StartSequence := FALSE;
b_ExtContactor := mode = eBreakerOperationMode.ExtGrid;
ton_ResetSEQ();

//SEQUENCER
CASE by_SequenceIndexes[ExecIndex] OF
	0: 	ExecIndex := 0; StartSequence := TRUE; by_RetryCounter := 0; by_CurrentStep := 0;
	1:	ton_ResetSEQ.IN := FALSE; by_CurrentStep := 1;
		b_trigger := Warmup(get.b_gensetHot);
	2:  b_trigger := SEL(b_ExtContactor, Inputcontactor.Close(b_SynchroneGenset OR b_GridFollowingMode), Extcontactor.Close(FALSE));
		get.e_state := eGenGridState.Synchronization; by_CurrentStep := 2;
		ton_ResetSEQ.IN := TRUE;
	3:	b_trigger := b_escapeCondition; by_CurrentStep := 3;
		get.e_state := eGenGridState.Starting;
END_CASE

ton_SeqPulse(IN := b_trigger AND NOT ton_SeqPulse.Q);
IF ton_SeqPulse.Q THEN
	ExecIndex := ExecIndex +1;
END_IF

IF ton_ResetSEQ.Q THEN
	ExecIndex := 0;
	ton_ResetSEQ.IN := FALSE;
	by_RetryCounter := by_RetryCounter + 1;
END_IF

IF by_RetryCounter > st_params.by_SyncRetries THEN
	by_RetryCounter := 0;
	get.events.b_WarmupFault := by_CurrentStep = 1;
	get.events.b_SynchronisationFault := by_CurrentStep = 2;
	get.events.b_StartupFault := by_CurrentStep = 3;
END_IF

//The exit from the current step. if breaker already closed, continue normal SFC procedure.
IF b_genOnly AND NOT b_startcondition AND NOT b_BreakerFb THEN
	b_IOStartStop := FALSE;
	SFCreset := TRUE;
END_IF
END_METHOD

METHOD StartStopConditions
VAR_INPUT
	enable			: BOOL;
END_VAR

VAR_INST
	r_LoadPercentOutput : REAL;
	b_Charging			: BOOL;
	r_InverterLoad		: REAL;
	r_InputLoad			: REAL;
	b_BatErrorGenStartTrigger : BOOL;
END_VAR
b_Charging:= monitor.powerstack.r_ActivePower < 0;
r_InverterLoad := monitor.powerstack.r_LoadPercent * SEL(b_Charging, 1, -1) * 0.97;// * monitor.system.r_CurrentEfficiency/100;
r_InputLoad	:= monitor.powermonitor.InputField.r_loadshare;
r_LoadPercentOutput := r_InputLoad + r_InverterLoad;

IF enable THEN
	ChargeLoadStart(
		enable:= b_loadbankEnable,
		reset := FALSE,
		value:= monitor.powerstack.r_LoadPercent, 
		startvalue:= MIN(GensetSetpoints.r_BatteryloadStart, monitor.powerstack.r_OvercurrentValueAct *100),
		stopvalue := GensetSetpoints.r_BatteryloadStop - monitor.powermonitor.InputField.r_loadshare,
		OffDelay := T#3M,
		OnDelay := T#10S);
	
	LoadStart(
		enable := monitor.powerstack.b_ControlEnabled,
		reset := r_LoadPercentOutput < -10,// if charging reset.
		value := r_LoadPercentOutput,
		StartValue:= MIN(GensetSetpoints.r_BatteryloadStart, monitor.powerstack.r_OvercurrentValueAct *100),
		StopValue :=  GensetSetpoints.r_BatteryloadStop,
		OffDelay := St_params.Genset.OverloadOffDelay,
		OnDelay := St_params.Genset.OverloadOnDelay,
		);
	
	SoCStart(
		enable := monitor.system.e_State <> eSystemState.Discharging_Only,
		reset := FALSE,
		value := monitor.battery.BatteryInfo.r_SOCScaled,
		StartValue:=  GensetSetpoints.r_SocStart,
		StopValue :=  MAX(GensetSetpoints.r_SocStop, GensetSetpoints.r_SocStart + 0.5));
		
	BatFullStart(
		enable:= b_loadbankEnable,
		reset := monitor.powerstack.r_ActivePower < -5 AND NOT b_loadbankEnable,
		value := monitor.battery.BatteryInfo.r_SOCScaled,
		StartValue:=  control.SoftSettings.system.r_SocMax,
		StopValue :=  control.SoftSettings.system.r_SocMax - settings.MachineParams.BMS.r_SocHysteresis,
		OffDelay := T#3M,
		OnDelay := T#10S
		);


ELSE
	BatFullStart(reset:= TRUE);
	SoCStart(reset := TRUE);
	LoadStart(reset := TRUE);
	ChargeLoadStart(reset := TRUE);
END_IF

//Trigger genset start when battery down.
IF NOT gensetsetpoints.b_StartAtBatteryError OR b_BESSready	THEN
	b_BatErrorGenStartTrigger := FALSE;
ELSIF NOT b_startcondition THEN
	b_BatErrorGenStartTrigger := TRUE;
END_IF

//Summerize conditions
b_StartCondition := ((LoadStart.Q OR SOCStart.Q OR BatFullStart.Q OR ChargeLoadStart.Q OR b_BatErrorGenStartTrigger) AND
						get.e_GensetStartStop= eGensetStartStop.Auto) OR 
						get.e_GensetStartStop= eGensetStartStop.Start;

//get run condition
IF get.e_GensetStartStop= eGensetStartStop.Start THEN
	get.e_RunCondition := eRunCondition.ManuallyStarted;
ELSIF get.e_GensetStartStop= eGensetStartStop.stop THEN
	get.e_RunCondition := eRunCondition.ManuallyStopped;
ELSIF SOCStart.Q THEN
	get.e_RunCondition := eRunCondition.SoC;	
ELSIF LoadStart.Q THEN
	get.e_RunCondition := eRunCondition.DischargeOverload;
ELSIF ChargeLoadStart.Q THEN
	get.e_RunCondition := eRunCondition.ChargeOverload;
ELSIF BatFullStart.Q THEN
	get.e_RunCondition := eRunCondition.BattFull;
ELSE
	get.e_RunCondition := eRunCondition.None;
END_IF
END_METHOD

ACTION STARTUP_active:
get.e_state := eGenGridState.Starting;
b_SFCmodetransInhibit := FALSE;
get.b_active := TRUE;


SFCtip := StartSequence(
			mode := BreakerOperationMode, 
			b_breakerfb := b_breakerFb,
			b_AcOK	:= b_BreakerACok,
			b_gridfollowingMode := b_GridACDetected,
			SFCreset => SFCResetTrigger
			) AND NOT sfctip;

//Reset before running again.		
GenDownCheck(FALSE, TRUE);
END_ACTION

ACTION STOP_active:
get.e_state := eGenGridState.Stopping;
SFCtransTrigger.in := FALSE;

CASE BreakerOperationMode OF
	eBreakerOperationMode.GenFix:
		IF Cooldown(TRUE) THEN SFCTransTrigger.in := InputContactor.Open(FALSE); END_IF
	eBreakerOperationMode.GenIso, eBreakerOperationMode.GenDroop:
	IF GenDownCheck(FALSE, FALSE) OR NOT b_breakerACOK THEN
		SFCTransTrigger.in := Inputcontactor.Open(TRUE) AND cooldown(TRUE);
	ELSIF NOT b_hybridMode AND b_startCondition AND monitor.powerstack.b_ControlEnabled AND NOT Get.b_ModeTransActive THEN
		InputContactor.Deload(TRUE);
		SFCTransTrigger.in := TRUE;
	ELSE
		SFCTransTrigger.in := InputContactor.Open(b_hybridMode) AND_THEN Cooldown(FALSE);
	END_IF
		
	eBreakerOperationMode.GridFeedthrough:
		IF b_AMFEnabled AND monitor.powerstack.b_ControlEnabled OR get.b_ModeTransActive THEN SFCTransTrigger.in := inputcontactor.Open(NOT Get.b_ModeTransActive OR get.events.b_CurrentLimitTrip);
		ELSE SFCTransTrigger.in := TRUE; END_IF
	eBreakerOperationMode.ExtGrid: 
		IF b_AMFEnabled AND monitor.powerstack.b_ControlEnabled THEN SFCTransTrigger.in := extcontactor.Open(control.SoftSettings.PSB.b_BreakerControl);
		ELSE SFCTransTrigger.in := TRUE; END_IF
END_CASE



SFCtip := SFCTransTrigger.Q AND NOT SFCtip;
END_ACTION

METHOD ThreePointSelector : REAL
VAR_INPUT
	r1max	: REAL;
	r2      : REAL;
	r3      : REAL;
	b2		: BOOL;
	b3		: BOOL;
END_VAR

VAR
	temp	: REAL;
END_VAR
IF b2 AND NOT b3 THEN
	temp := r2;
ELSIF NOT b2 AND b3 THEN
	temp := r3;
ELSE
	temp := r1max;
END_IF

ThreepointSelector := LIMIT(0,temp,r1max);
END_METHOD

ACTION WAITINGTRIGGER_active:
get.e_state := eGenGridState.Waiting_Trigger;
SFCTransTrigger.IN := FALSE;
get.b_active := FALSE;

CASE BreakerOperationMode OF
	eBreakerOperationMode.GenIso:
		SFCTransTrigger(IN := b_StartCondition AND NOT GenDownCheck(FALSE , b_StartCondition));
	eBreakerOperationMode.GenDroop:
		SFCTransTrigger(IN := b_StartCondition AND NOT GenDownCheck(FALSE , b_StartCondition)); 
	eBreakerOperationMode.Genfix:
		SFCTransTrigger(IN := b_StartCondition AND NOT GenDownCheck(FALSE , b_StartCondition) AND b_BESSReady AND b_BusbarACOK);
	eBreakerOperationMode.Gridfeedthrough, eBreakerOperationMode.ExtGrid: 
		SFCTransTrigger(IN := b_breakerACOK);
		get.e_state := eGenGridState.Waiting_For_AC;
		IF NOT GridOKdetect(FALSE) THEN
			get.e_state := eGenGridState.Gridcode_Release_Check;
			SFCTransTrigger.in := FALSE;
		END_IF
END_CASE

IF get.b_ModeTransActive THEN
	get.e_state := eGenGridState.Waiting_Mode_Reconnect;
END_IF

IF b_ForceOperate OR (b_breakerfb AND b_breakerACOK) THEN
	SFCTransTrigger.in := TRUE;
END_IF



//Trigger to start. Only if modeswitch is disabled.
SFCtip := SFCTransTrigger.Q AND NOT get.b_ModeTransActive AND NOT SFCtip AND NOT get.events.b_StartingInhibit;
END_ACTION

METHOD Warmup : BOOL
VAR_INPUT
	Skip		: BOOL;
END_VAR

VAR_INST
	t_time				: TIME;
	b_startfb			: BOOL;
	ton_StartTimeOut	: TON;
	tof_reset			: Tof := (PT:= T#20MS);
END_VAR
b_IOStartStop := TRUE;
Warmup := FALSE;

b_startFb := b_BreakerACok;
IF NOT b_breakerACOK THEN
	inputcontactor.open(TRUE);
	get.e_state := eGenGridState.Starting;
ELSE
	get.e_state := eGenGridState.Warmup;
END_IF

tof_reset(IN:= NOT ton_StartTimeOut.Q);
ton_StartTimeOut(IN := b_startfb AND tof_reset.Q, PT:= t_WarmupTime); 

IF ton_StartTimeOut.Q OR skip THEN
	get.b_gensetHot := TRUE;
	ton_StartTimeOut.IN := FALSE;
	Warmup := b_IOStartStop;
END_IF
END_METHOD

METHOD ZeroCurrentDisconnect : BOOL
VAR_INPUT
END_VAR

VAR_INST
	ton_FlatZeroCurrentTimeOut 	: TON := (PT:= T#50MS);
END_VAR
ton_FlatZeroCurrentTimeOut(
	IN := TO_INT(ar_BreakerCurrent[phases.L1]) = 0 OR TO_INT(ar_BreakerCurrent[phases.L2]) = 0 OR TO_INT(ar_BreakerCurrent[phases.L3]) = 0,
	Q => ZeroCurrentDisconnect);
END_METHOD

END_FUNCTION_BLOCK

// ---- POUs/System/GenGridControl/FB_ContactorControl.TcPOU
FUNCTION_BLOCK FB_ContactorControl
VAR_IN_OUT CONSTANT
	monitor								   	: ST_System_Monitor;
	control									: ST_System_Control;
	st_params								: ST_ContactorControl_params;
END_VAR

VAR_IN_OUT
	SyncData								: ST_GenGridController_SyncData;

END_VAR

VAR_INPUT
	b_fbIn			: BOOL;
	b_deadbus		: BOOL;
	b_SyncOK		: BOOL;
	li_VoltCrossRef	: LINT;
	li_VoltCrossBus	: LINT;
	r_AcVoltageRef	: REAL;
	r_AcFreqRef		: REAL;
	e_AcRotationRef : eACRotationState; // Fsource of reference
	e_AcRotationBus	: eACRotationState; //bus 
	ar_current		: ARRAY [0..4] OF REAL;
	r_power			: REAL;	
	b_deloadEnable	: BOOL;
END_VAR
VAR_OUTPUT
	CloseCMD		: BOOL;
	OpenCMD			: BOOL;
	SyncEnable		: BOOL;
	FreqSet			: REAL;
	VoltSet			: REAL;
	ACok			: BOOL;	
	b_fb			: BOOL;
	b_Deload		: BOOL;
	RotationFault	: BOOL;
END_VAR

VAR
	ton_SyncDelay 	: TON := (PT:=  T#1S);
	
	ton_synccheckoffdelay : TON := (PT :=T#1s);
	SyncCheck		: BOOL;
	fb_VoltPID			: FB_CTRL_PID_EXT;
	st_Params_VoltPID				: ST_CTRL_PID_EXT_PARAMS := ( 
										tTaskCycleTime := T#1MS,
										tCtrlCycleTime := T#1MS,
										fKp	:= 0.3,
										tTn := T#200MS,
										tTd := T#0MS,
										tTv := T#0MS,
										fOutMaxLimit := 40,
										fOutMinLimit := -40										
);
END_VAR

ACok := ACcheck(r_voltage := r_ACVoltageRef, r_frequency := r_ACFreqRef);
CheckRotationField();
SyncEnable := syncdata.b_Sync OR SyncCheck;
ton_SyncDelay(IN := SyncEnable);
b_fb := b_fbIn;

fb_VoltPID(stParams := st_Params_VoltPID);
ton_synccheckoffdelay(IN:= b_fb);
IF ton_synccheckoffdelay.Q THEN
	synccheck := FALSE;
	fb_VoltPID.eMode:= e_Ctrl_mode.eCTRL_MODE_RESET;
END_IF

METHOD CheckRotationField : BOOL
VAR_INPUT
END_VAR
IF e_ACRotationRef <> 0 AND e_ACRotationBus <> 0 THEN // if both are connected to AC
	IF e_ACRotationRef = e_ACRotationBus THEN
		CheckRotationField := TRUE;
		RotationFault := FALSE;
	ELSE
		RotationFault := TRUE;
	END_IF
ELSE
	RotationFault := FALSE;
END_IF
END_METHOD

METHOD Close : BOOL
VAR_INPUT
	Force	: BOOL;
END_VAR
VAR_INST
	ton_ACOKrelease : TON := (PT:= T#1S); 
	b_VoltageDetected	: BOOL;
	
	ton_SyncOK			: TON := (PT := T#5S);
END_VAR
ton_ACOKrelease(IN:= ACok);
b_VoltageDetected := r_ACVoltageRef > 100;
OpenCMD := FALSE;
syncCheck := FALSE;

ton_SyncOK(IN :=b_syncOK);
IF b_fbIN OR b_deadbus THEN
	CloseCMD := TRUE;
ELSIF force THEN
	IF b_VoltageDetected AND NOT b_deadbus THEN
		syncCheck := TRUE;
		CloseCMD := ton_SyncOK.Q AND ton_ACOKrelease.Q;
	ELSE
		CloseCMD := TRUE;
	END_IF
ELSE
	CloseCMD:= Sync();
END_IF

Close := b_fbIN;
IF b_fbIN THEN
	Syncdata.b_Sync := FALSE;
	syncCheck := FALSE;
	ton_SyncOK.IN := FALSE;
	ton_ACOKrelease.IN :=  FALSE;
END_IF
END_METHOD

METHOD Deload : BOOL
VAR_INPUT
	reset : BOOL;
END_VAR

VAR_INST
	release : BOOL;
	PowerReleaseThreshold : REAL;
	
END_VAR
IF b_deloadEnable AND NOT reset THEN
	b_Deload := TRUE;
	PowerReleaseThreshold := st_params.ui_DeloadCurrentRelease * r_AcVoltageRef *  1.73 / 1000; 
	release := ABS(ar_current[0]) < st_params.ui_DeloadCurrentRelease OR ABS(r_power) < (PowerReleaseThreshold);
	IF release THEN
		Deload := TRUE;
	END_IF
ELSE
    b_Deload := FALSE;
	Deload := TRUE;
END_IF
END_METHOD

METHOD FreqControlPID : BOOL;
VAR_INPUT
	r_ACRef				: REAL;
	r_ACintern			: REAL;
END_VAR

VAR_OUTPUT
	Q					: REAL;
END_VAR


VAR_INST
	r_phaseTimeDelta		: REAL;
	r_PeriodTime			: REAL;
	r_phaseAngle			: REAL;
	Buffer  				: ARRAY[0..2] OF REAL;
    Index   				: UINT := 0;
	di_tempAngle			: DINT;
	r_phaseAngleEMA        	: REAL := 0.0; // startwaarde
    Alpha       			: REAL := 0.5; // dempingsfactor tussen 0 en 1
	
		fb_FreqPID						: FB_CTRL_PID_EXT;
		st_Params_FreqPID				: ST_CTRL_PID_EXT_PARAMS := ( 
										tTaskCycleTime := T#1MS,
										tCtrlCycleTime := T#1MS,
										fKp	:= 0.1,
										tTn := T#20MS,
										tTd := T#0MS,
										tTv := T#0MS,
										fOutMaxLimit := 0.03,
										fOutMinLimit := -0.03										
);
	ton_SyncOKdelay						: TON := (PT := T#1S);
	r_syncOKAngle						: REAL := 2.0;
	r_FreqOffset 						: REAL := -0.05;
	
	li_voltcrossbusLast					: LINT;
	li_VoltCrossRefLast					: LINT;
	ton_FreqPIDBypass					: TON := (PT := T#2S);
	
END_VAR
ton_FreqPIDBypass(IN := li_voltcrossbusLast = li_voltcrossbus OR li_VoltCrossRefLast = li_VoltCrossRef);
IF ton_FreqPIDBypass.Q THEN
	 r_freqOffset := -0.05;
	 ton_SyncOKdelay(IN := b_syncOK, PT:= T#0S);
ELSE
	r_PeriodTime := SEL(r_ACintern = 0, 1/r_ACintern, 0) * 1000;
	r_phaseTimeDelta := TO_REAL((li_VoltCrossbus - li_VoltCrossRef) MOD TO_DINT(r_PeriodTime*1000000)) /1000000;
	
	IF r_phaseTimeDelta > (r_PeriodTime /2)  THEN
		r_phaseTimeDelta := r_phaseTimeDelta - r_PeriodTime; 
	ELSIF r_phaseTimeDelta < -(r_PeriodTime /2) THEN
		r_phaseTimeDelta := r_phaseTimeDelta + r_PeriodTime; 
	END_IF
	
	// Stap 1: bereken eerst de DINT-waarde veilig
	di_tempAngle := TO_DINT(r_phaseTimeDelta * r_ACintern * 360);
	
	// Stap 3: schaal naar REAL
	r_phaseAngle := TO_REAL(di_tempAngle MOD 360000) / 1000;
	
	//setup filtering (median and exponential moving average)
	Buffer[Index MOD 3] := r_phaseAngle;
	Index := Index + 1;
	r_phaseAngleEMA := Alpha * median(buffer) + (1.0 - Alpha) * r_phaseAngleEMA;
	
	fb_FreqPID(
		fSetpointValue := 0,
		fActualValue :=  r_phaseAngleEMA,
		stParams:= st_Params_FreqPID,
		fout => r_FreqOffset);
		
	fb_FreqPID.bHold := r_phaseAngleEMA > 170 OR r_phaseAngleEMA < -170;
	
		
	IF NOT fb_FreqPID.bError THEN
		fb_FreqPID.eMode := e_CTRL_MODE.eCTRL_MODE_ACTIVE;
	ELSE
		fb_FreqPID.eMode := e_CTRL_MODE.eCTRL_MODE_RESET;
	END_IF
	
	ton_SyncOKdelay(IN := ABS(r_phaseAngleEMA) < r_syncOKAngle, PT:= T#2S);
END_IF

//set outputs
Q := r_ACRef - r_freqOffset;
FreqControlPID := ton_SyncOKdelay.Q;


//update on change values
li_voltcrossbusLast := li_voltcrossbus;
li_voltcrossrefLast := li_voltcrossref;
END_METHOD

METHOD FrequencyControl : BOOL
VAR_INPUT
	r_ACRef				: REAL;
	r_ACintern			: REAL;
END_VAR

VAR_OUTPUT
	Q					: REAL;
END_VAR


VAR_INST
	OK					: BOOL;
	r_FreqOffset 		: REAL := 0.1; // hz
END_VAR
//Go below ref Frequency.

Q := r_ACRef + r_FreqOffset;
OK := ABS(r_ACintern - r_ACRef) < ABS(4* r_FreqOffset);
FrequencyControl := OK;
END_METHOD

METHOD init : BOOL
VAR_INPUT
END_VAR
syncCheck := FALSE;
END_METHOD

METHOD Open : BOOL
VAR_INPUT
	b_force : BOOL;
END_VAR

VAR_INST
	ton_TimeOut : TON;
END_VAR
ton_TimeOut(PT := TO_TIME(TO_REAL(st_params.ui_DeloadTimeOut)*1000));
CloseCMD := FALSE;

IF b_force OR ton_timeOut.Q THEN
	OpenCMD := TRUE;
ELSE
	ton_TimeOut.IN := TRUE;
	OpenCMD := Deload(FALSE);
END_IF

open := NOT b_FbIN;
IF NOT b_fbIn THEN
	//Syncdata.b_Sync:= FALSE;
	ton_TimeOut.IN := FALSE;
	b_deload := FALSE;
	OpenCMD := FALSE;
END_IF
END_METHOD

METHOD PRIVATE Sync : BOOL

VAR_INST
	//OK : BOOL;
	phasecontrol : BOOL := FALSE;
	SyncOKSum	: BOOL;
	tp_SyncOK : TP := (PT := T#100MS);
END_VAR
Syncdata.b_Sync := ACok;

IF phasecontrol THEN //new method beckhoff phase matching
	SyncOKsum := FreqControlPID(r_ACFreqRef, monitor.powerstack.r_FrequencyD7, Q => Syncdata.r_freqSet);
ELSE //old method
	SyncOKSum := b_syncOK AND FrequencyControl(r_acRef := r_ACFreqRef,  r_ACintern := monitor.powerstack.r_FrequencyD7, Q => Syncdata.r_freqSet);
END_IF

tp_SyncOK(IN:= SyncOKsum AND
	ACok AND
	CheckRotationField() AND
	VoltageControl(r_acRef := r_ACvoltageRef, r_ACintern := monitor.powerstack.r_ACVoltageD7, Q => Syncdata.r_VoltSet)
	);

IF ton_SyncDelay.Q AND tp_SyncOK.Q THEN
	SyncOKSum := FALSE;
	Sync := TRUE;
END_IF
END_METHOD

METHOD VoltageControl : BOOL
VAR_INPUT
	r_ACRef				: REAL;
	r_ACintern			: REAL;
END_VAR
VAR_OUTPUT
	Q : REAL;
END_VAR

VAR_INST
	
	OK			: BOOL;
	VoltDev		: REAL;

END_VAR
//Go equal to ref voltage.
VoltDev := r_ACintern - r_ACRef; 

//TOTAL AC CURRENT LIMIT
st_Params_VoltPID.fInnerWindow :=  st_Params.VoltagePID.InnerWindow;
st_Params_VoltPID.fOuterWindow := st_Params.VoltagePID.OuterWindow;
st_Params_VoltPID.fKp := st_params.VoltagePID.Kp;
st_Params_VoltPID.tTn := TO_TIME(st_params.VoltagePID.Tn);
st_Params_VoltPID.tTd := TO_TIME(st_params.VoltagePID.Td);
st_Params_VoltPID.tTv := TO_TIME(st_params.VoltagePID.Tv);
st_params_VoltPID.fDeadBandInput := st_Params.VoltagePID.InputDeadband;
st_params_VoltPID.fDeadBandOutput := st_Params.VoltagePID.OutputDeadband;

fb_VoltPID.fActualValue := VoltDev;
	
IF st_Params.VoltagePID.enable THEN
	fb_VoltPID.eMode := e_CTRL_MODE.eCTRL_MODE_ACTIVE;
ELSE
	fb_VoltPID.eMode := e_CTRL_MODE.eCTRL_MODE_RESET;
END_IF
	
OK := ABS(VoltDev) < st_params.ui_VoltageDevSyncOK;
Q := r_ACRef + fb_VoltPId.fOut;
VoltageControl := OK;
END_METHOD

END_FUNCTION_BLOCK

// ---- POUs/Functions-FBs-Programs/_acFunctions/AcCheck.TcPOU
FUNCTION AcCheck : BOOL
VAR_INPUT
	r_Voltage	: REAL;
	r_Frequency	: REAL;
END_VAR

AcCheck	:= AcFrequencyCheck(r_Frequency) AND AcVoltageCheck(r_Voltage);

END_FUNCTION

// ---- POUs/Functions-FBs-Programs/_acFunctions/ACFrequencyCheck.TcPOU
FUNCTION ACFrequencyCheck : BOOL
VAR_INPUT
	IN			: REAL;
END_VAR
VAR
	r_min		: REAL;
	r_max		: REAL;
END_VAR

r_min:= settings.GridParams.r_GridFrequencyMin;
r_max:= settings.GridParams.r_GridFrequencyMax;

ACfrequencyCheck := LIMIT(r_min, IN, r_max) = IN;

END_FUNCTION

// ---- POUs/Functions-FBs-Programs/_acFunctions/ACVoltageCheck.TcPOU
FUNCTION ACVoltageCheck : BOOL
VAR_INPUT
	IN			: REAL;
END_VAR
VAR
	r_min		: REAL;
	r_max		: REAL;
END_VAR

r_min:= settings.GridParams.r_GridVoltageMin - 10;
r_max:= settings.GridParams.r_GridVoltageMax;

ACVoltageCheck := LIMIT(r_min, IN, r_max) = IN;

END_FUNCTION

// ---- POUs/Functions-FBs-Programs/_generalFunctions/Median.TcPOU
FUNCTION Median : REAL
VAR_IN_OUT
    arr : ARRAY[*] OF REAL;
END_VAR

VAR
    sorted : ARRAY[0..6] OF REAL;
    i, j   : INT;
    temp   : REAL;
    len    : INT;
END_VAR



// bepaal lengte
len := TO_INT(UPPER_BOUND(arr, 1) - LOWER_BOUND(arr, 1) + 1);

// safety check
IF len > 7 THEN
    len := 7;
END_IF

// kopie
FOR i := 0 TO len - 1 DO
    sorted[i] := arr[i + LOWER_BOUND(arr,1)];
END_FOR

// sort
FOR i := 0 TO len - 2 DO
    FOR j := 0 TO len - i - 2 DO
        IF sorted[j] > sorted[j + 1] THEN
            temp := sorted[j];
            sorted[j] := sorted[j + 1];
            sorted[j + 1] := temp;
        END_IF
    END_FOR
END_FOR

// median
IF (len MOD 2) = 0 THEN
    Median := (sorted[len/2 - 1] + sorted[len/2]) * 0.5;
ELSE
    Median := sorted[len/2];
END_IF

END_FUNCTION

// ---- POUs/Functions-FBs-Programs/_generalFunctions/FB_StartStop.TcPOU
FUNCTION_BLOCK FB_StartStop
VAR_INPUT
	enable : BOOL;
	reset: BOOL;
	value : REAL;
	StartValue : REAL;
	StopValue : REAL;
	GreaterThan	: BOOL;
	OffDelay	: TIME;
	OnDelay		: TIME;	
END_VAR
VAR_OUTPUT
	Q : BOOL;
END_VAR
VAR
	SR_Started : SR;
	ton_set : TON;
	ton_reset: TON;
	ton_minruntime : TON;
END_VAR

ton_set(PT := Ondelay);
ton_reset(PT := Ondelay);
ton_minruntime(PT := OffDelay);
SR_Started();

IF GreaterThan THEN
	ton_set.IN:= value >= StartValue AND NOT reset;
	ton_reset.IN:= value <= StopValue OR reset;
ELSE
	ton_set.IN:= value <= StartValue AND NOT reset;
	ton_reset.IN:= Value >= StopValue OR reset;
END_IF

ton_minruntime(IN:= sr_started.Q1);
IF enable THEN
	SR_Started.SET1 := ton_set.Q;
	SR_Started.RESET := ton_reset.Q AND ton_minruntime.Q;
	Q := sr_started.Q1;	
ELSE
	SR_Started.SET1 := FALSE;
	SR_Started.RESET := TRUE;
	Q := FALSE;
END_IF

END_FUNCTION_BLOCK

// ---- POUs/Functions-FBs-Programs/_generalFunctions/PackWord.TcPOU
FUNCTION PackWord : WORD
VAR_INPUT
	b0			: BOOL;
	b1			: BOOL;
	b2			: BOOL;
	b3			: BOOL;
	b4			: BOOL;
	b5			: BOOL;
	b6			: BOOL;
	b7			: BOOL;
	b8			: BOOL;
	b9			: BOOL;
	b10			: BOOL;
	b11			: BOOL;
	b12			: BOOL;
	b13			: BOOL;
	b14			: BOOL;
	b15			: BOOL;
END_VAR

PackWord.0	:= b0;
PackWord.1	:= b1;
PackWord.2	:= b2;
PackWord.3	:= b3;
PackWord.4	:= b4;
PackWord.5	:= b5;
PackWord.6	:= b6;
PackWord.7	:= b7;
PackWord.8	:= b8;
PackWord.9	:= b9;
PackWord.10	:= b10;
PackWord.11	:= b11;
PackWord.12	:= b12;
PackWord.13	:= b13;
PackWord.14	:= b14;
PackWord.15	:= b15;

END_FUNCTION

// ---- POUs/Objects/ACDCCharger/FB_AcDcCharger.TcPOU
FUNCTION_BLOCK FB_AcDcCharger

VAR_IN_OUT CONSTANT
	st_params				:	ST_ACDCCharger_Params;
END_VAR

VAR_IN_OUT
	st_service : ST_ACDCCharger_Service;
END_VAR

VAR_INPUT
	enable					: 	BOOL;

	Set						:	ST_ACDCCharger_set;
	//BMS					:	st_BMS_BatterySummary;	
	r_Soc 					: 	REAL;
	r_SystemVoltage			: 	REAL;
	r_SystemCurrent			: 	REAL;
	r_MaxChargeCurrent		:	REAL;
	b_BatteryFullyCharged	: BOOL;
	b_BatteryOn				: BOOL;	
END_VAR
VAR_OUTPUT
	Get			:	ST_ACDCCharger_get;
	IPSRequest	:	ST_InternalPowerSupply_PowerDemand;
END_VAR
VAR
	BuscouplerState	AT %I*	: UINT;
	RxQueue			AT %I*	:	CANRXQUEUESTRUCT_E_10;  //without Transaction Time
	TxQueue			AT %Q*	:	CANTXQUEUESTRUCT_E_10;
	b_BuscouplerFound: BOOL;
END_VAR
VAR   // should add as input var
    bEmergencyStop : BOOL := FALSE;
    bResetFault : BOOL;
	GroupID	: BYTE := 1;
//	uiNumberofUnits	: UINT :=1;  // the number of units that are phyzicaly designed
//	rPset	: REAL; // AC Power set limit
//	rIset   : REAL; // AC Current set limit
//	bPowerMode : BOOL; // P mode sett selection
END_VAR
VAR	
	diag 	: ST_SystemDiagnostic;
    txIndex : INT;
    Step 	: INT;
    NumberOfMessagesToSend : INT := 10;

    voltage_mV : UDINT;
    current_mA : UDINT;
	stData : ST_Data;
    stControl : ST_Control;
	DeviceNo   : BYTE := 16#0B;
	rxIndex : INT; 
//    ChargerState : E_ChargerState := E_ChargerState.Idle;
	rVoltageWindow : REAL := 5.0;   // should be base on percentage or Volt?!
    bVoltageWindowOk : BOOL;  // check if voltage within the window
    b_ModuleCommunicationLost : BOOL;
    bWarning : BOOL;
    rChargerVoltageSetpoint : REAL;
    rChargerCurrentSetpoint : REAL;
    eval : ST_SystemEval;	
	bValidPrev : ARRAY [0..10] OF BOOL;  // test
	bFreezeCurrent : BOOL; // test	
	rMaxLimit		: REAL;

    tCycle : TON;
    tCheck : TON;
    tComWatchdog : TON;
    rPower_kW : REAL;
    rIsetReq : REAL := 60.0; (* configurable *)
    rCurrentCmd : REAL;
END_VAR
VAR CONSTANT
	e_ID 				: eObject_ID := eObject_ID.ACDCCharger;
END_VAR


IF enable THEN
	IF (BuscouplerState <> 8) THEN
		get.e_SystemStatus := eACDCChargerstate.init;
		get.Events.b_BuscouplerNotFound := TRUE;
	ELSE
		get.Events.b_BuscouplerNotFound := False;
		IF get.e_SystemStatus = eACDCChargerstate.init THEN
			get.e_SystemStatus := eACDCChargerstate.off;
		END_IF
		
		// should be 50ms to 200ms 
		tCycle(IN := NOT tCycle.Q, PT := T#50MS);
				
		IF tCycle.Q THEN
			ReadingRx();
			//UpdateStData();  // keep the last value! Useless?!
			EvaluateSystem();
			ChargingControl();
			SafetyCheck();
		    ValidateOutput();
			RunStateMachine();
			HandleCanCommunication();
			EvaluateDiagnostics();
		END_IF
	END_IF
END_IF

METHOD BuildCanId : DWORD
VAR_INPUT
    CommandNo  : BYTE;   // protocol command
    TargetAddr : BYTE := 1;   // group / module / broadcast(0x3F)
	
END_VAR
VAR
	 ErrorCode : BYTE := 0;   // always 0
	 SourceAddr : BYTE := 16#F0;   // Controller address
END_VAR

  // TargetAddr := 1;
   DeviceNo := 16#0B;
   ErrorCode:= 0;
   SourceAddr := 16#F0;
   
   
   BuildCanId :=
      SHL(DWORD#1,31)                // bit31 = extended CAN frame
   OR SHL(TO_DWORD(ErrorCode),26)       // error code
   OR SHL(TO_DWORD(DeviceNo),22)        // device number   Multicas: 0x0B, BroadCasti:0x0A
   OR SHL(TO_DWORD(CommandNo),16)       // command 
   OR SHL(TO_DWORD(TargetAddr),8)       // target address
   OR TO_DWORD(SourceAddr);             // source address
END_METHOD

METHOD PRIVATE ChargingControl
VAR_INPUT
END_VAR
VAR_INST
	rRawV : REAL;
	rPrevV : REAL;
	rRampLimitV : REAL := 20;
	rCurrentReq : REAL;
	rVoltageRamp : REAL;
	rAcPower	: REAL;
	rAcCurrent : REAL := 0.0;
	rMinGridVoltage	: REAL;
	i : INT;
	rTempMin : REAL;
	tDelayJumpOff	: TOf;
	bTestb : BOOL;
	srTest	: SR;
	tTestB : TOF;
	iUnitsTemp	: INT;
	
	iPrevHealthyModules : INT;
	tNewModuleTimer : TON;
	iEffectiveModules : INT;
	
	rTest : REAL;
	
	r_MinGridVoltageDerating 	: REAL := 1;
	r_TempDerating 				: REAL := 1;
	BMSChargeCurrentLimit		:	REAL;
	
	
END_VAR
 
// Battery Voltage from BMS

set.r_MinGridVoltage 	:= LIMIT(360, set.r_MinGridVoltage, 440);
set.r_currentSetpoint 	:= LIMIT(0, set.r_currentSetpoint, 125);
set.r_powersetpoint 	:= LIMIT(0, set.r_powersetpoint, st_params.ui_ModuleDesignPower * st_params.ui_NrOfInstalledModules);
set.r_SocTarget 		:= LIMIT(0, set.r_SocTarget, 100);

IF b_BatteryOn THEN // bms.e_BMS_PowerOnStatus = ePowerOnSTatus.On THEN
	rChargerVoltageSetpoint := r_SystemVoltage + st_params.r_VoltageWindow;
ELSE
	rChargerVoltageSetpoint := 0.0;
END_IF

IF r_Soc >= set.r_SocTarget OR b_BatteryFullyCharged THEN//bms.e_BMS_Status = eBMS_status.FullCharge THEN
	get.events.b_SOCLimitReached := TRUE;
ELSIF r_Soc < set.r_SocTarget - st_params.SocHysteresis THEN
	get.events.b_SOCLimitReached := FALSE;
END_IF


//rPower_kW := (stData.rSystemOutVoltageDc * stData.rSystemOutCurrentDc) / 1000.0;

rMinGridVoltage := 1000.0;
FOR i := 0 TO TO_INT(st_params.ui_NrOfInstalledModules - 1) DO
    IF stData.stModuleData[i].rExternalVoltageDc > 550 AND NOT stData.stModuleData[i].stStatus.bPfcOff  THEN
        
        rTempMin := MIN( stData.stModuleData[i].rVoltageL1L2,
            				stData.stModuleData[i].rVoltageL2L3,
            				stData.stModuleData[i].rVoltageL3L1 );
        
        rMinGridVoltage := MIN(rMinGridVoltage, rTempMin);        
    END_IF;
END_FOR;

IF (stData.rSystemOutVoltageDc > 1.0) THEN
	CASE set.e_ControlType OF
		ePowerControlType.Power		:	
			rIsetReq := (set.r_powersetpoint * 1000 / stData.rSystemOutVoltageDc) * 0.95;
			get.events.b_CurrentLimitActive := FALSE;
			
		ePowerControlType.Current 	:	
			rIsetReq := ((rMinGridVoltage * set.r_currentSetpoint * 1.73) / stData.rSystemOutVoltageDc) * 0.95;
			get.events.b_CurrentLimitActive := TRUE;
			
		ePowerControlType.Both 		:	
			rIsetReq := (set.r_powersetpoint * 1000 / stData.rSystemOutVoltageDc) * 0.95;
			IF (rMinGridVoltage * set.r_currentSetpoint * 1.73) < set.r_powersetpoint * 1000 THEN
				rIsetReq := ((rMinGridVoltage * set.r_currentSetpoint * 1.73) / stData.rSystemOutVoltageDc) * 0.95;
				get.events.b_CurrentLimitActive := TRUE;
			ELSE
				get.events.b_CurrentLimitActive := FALSE;
			END_IF
	END_CASE
ELSE
	riSetReq := 0;
END_IF

BMSChargeCurrentLimit := ABS(r_MaxChargeCurrent) + r_SystemCurrent + stData.rSystemOutCurrentDc;
IF BMSChargeCurrentLimit < rIsetReq THEN
	rCurrentCmd := BMSChargeCurrentLimit - 2;
	get.Events.b_BatteryLimitDeratingActive := TRUE;
ELSE
	rCurrentCmd := MIN(rCurrentCMD + ST_Params.BMSChargeLimitRampRate, rIsetReq);
	get.Events.b_BatteryLimitDeratingActive := FALSE;
END_IF

 
//ACVoltageRamp
IF rMinGridVoltage < set.r_MinGridVoltage THEN
	r_MinGridVoltageDerating := MAX(r_MinGridVoltageDerating * 0.999, 0.1);
ELSIF rMinGridVoltage > set.r_MinGridVoltage + st_params.GridVoltageHysteresis THEN
	r_MinGridVoltageDerating := MIN(r_MinGridVoltageDerating * 1.001, 1);
END_IF

get.Events.b_ACUnderVoltageDeratingActive := r_MinGridVoltageDerating < 1;


IF eval.rMaxTemperature > 80.0 THEN
	r_TempDerating := MAX(r_TempDerating * 0.999, 0.1);
ELSIF eval.rMaxTemperature < 75.0 THEN
	r_TempDerating := MIN(r_TempDerating * 1.001, 1);
END_IF
get.Events.b_TemperatureDeratingActive := r_TempDerating < 1;


// a unit back after a short lost( less than 10s  and keep stData.rNumberOfModules as original value)
iEffectiveModules := eval.iHealthyModules;
IF eval.iHealthyModules > iPrevHealthyModules THEN
	iEffectiveModules := eval.iHealthyModules + (eval.iHealthyModules - iPrevHealthyModules);
END_IF


// Current setpoint
//rCurrent := LIMIT(0.0, rCurrentCmd, eval.rTotalAvailableCurrent) / MAX(iEffectiveModules, 1);
IF bFreezeCurrent THEN
    rChargerCurrentSetpoint := 0;              // or keep last value if you prefer
    bFreezeCurrent := FALSE;    // only 1 cycle
ELSE
    rChargerCurrentSetpoint := LIMIT(0.0, rCurrentCmd, eval.rTotalAvailableCurrent) / MAX(iEffectiveModules, 1);
END_IF

iPrevHealthyModules := eval.iHealthyModules;

// if any unit is back after a long lost, stData.rNumberOfModules become 0 for a momment
tDelayJumpOff(IN := (stData.rNumberOfModules < eval.iHealthyModules), PT := T#1S);

IF tDelayJumpOff.Q THEN
	rChargerCurrentSetpoint := 0.0;
END_IF

IF iEffectiveModules > 0 THEN
	rChargerCurrentSetpoint := 
		LIMIT(0, rChargerCurrentSetpoint * r_MinGridVoltageDerating * r_TempDerating, eval.rTotalAvailableCurrent / iEffectiveModules);
ELSE
	rChargerCurrentSetpoint := 0;
END_IF
END_METHOD

METHOD EMSTOP : BOOL
VAR_INPUT
END_VAR


get.e_SystemStatus := eACDCChargerState.Fault;

EMSTOP := true;
END_METHOD

METHOD PRIVATE EvaluateDiagnostics
VAR
    i : INT;
END_VAR
	

//Reset all
diag.bAnyError 				:= FALSE;
diag.bAnyWarning 			:= FALSE;

diag.bError_OutputOV 		:= FALSE;
diag.bError_OverTemp 		:= FALSE;
diag.bError_ShortCircuit	:= FALSE;
diag.bError_ModuleError 	:= FALSE;
diag.bError_CommLost 		:= FALSE;
diag.bError_PhaseLost 		:= FALSE;

diag.bWarn_InputOV 			:= FALSE;
diag.bWarn_InputUV 			:= FALSE;
diag.bWarn_FanError 		:= FALSE;
diag.bWarn_PowerLimit 		:= FALSE;
diag.bWarn_TempHigh 		:= FALSE;

diag.bAllModulesOff 		:= TRUE;
diag.bAllModulesOn 			:= TRUE;


FOR i := 0 TO TO_INT(st_params.ui_NrOfInstalledModules - 1) DO

    //ERRORS
    IF stData.stModuleData[i].stStatus.bOutputOverVoltage THEN
        diag.bError_OutputOV := TRUE;
    END_IF

    IF stData.stModuleData[i].stStatus.bTempHigh THEN
        diag.bError_OverTemp := TRUE;
    END_IF

    IF stData.stModuleData[i].stStatus.bOutputShortCircuit THEN
        diag.bError_ShortCircuit := TRUE;
    END_IF

    IF stData.stModuleData[i].stStatus.bModuleError OR
       stData.stModuleData[i].stStatus.bModuleProtection THEN
        diag.bError_ModuleError := TRUE;
    END_IF

    IF stData.stModuleData[i].stStatus.bCanTimeout THEN
        diag.bError_CommLost := TRUE;
    END_IF

    IF stData.stModuleData[i].stStatus.bPhaseLost THEN
        diag.bError_PhaseLost := TRUE;
    END_IF


    //WARNINGS
    IF stData.stModuleData[i].stStatus.bInputOverVoltage THEN
        diag.bWarn_InputOV := TRUE;
    END_IF

    IF stData.stModuleData[i].stStatus.bInputUnderVoltage THEN
        diag.bWarn_InputUV := TRUE;
    END_IF

    IF stData.stModuleData[i].stStatus.bFanError THEN
        diag.bWarn_FanError := TRUE;
    END_IF

    IF stData.stModuleData[i].stStatus.bPowerLimitation THEN
        diag.bWarn_PowerLimit := TRUE;
    END_IF

    IF stData.stModuleData[i].stStatus.bTempHigh THEN
        diag.bWarn_TempHigh := TRUE;
    END_IF


    //MODULE STATE
    IF NOT stData.stModuleData[i].stStatus.bDcSideOff AND stData.stModuleData[i].stStatus.bSlowStartup THEN
        diag.bAllModulesOff := FALSE;
    END_IF

    IF stData.stModuleData[i].stStatus.bDcSideOff AND stData.stModuleData[i].stStatus.bSlowStartup THEN
        diag.bAllModulesOn := FALSE;
    END_IF

END_FOR

IF diag.bAllModulesOff THEN
	diag.bAllModulesOn := FALSE;
END_IF


//GLOBAL FLAGS
diag.bAnyError :=
    diag.bError_OutputOV OR
    diag.bError_OverTemp OR
    diag.bError_ShortCircuit OR
    diag.bError_ModuleError OR
    diag.bError_CommLost OR
    diag.bError_PhaseLost;

diag.bAnyWarning :=
    diag.bWarn_InputOV OR
    diag.bWarn_InputUV OR
    diag.bWarn_FanError OR
    diag.bWarn_PowerLimit OR
    diag.bWarn_TempHigh;
END_METHOD

METHOD PRIVATE EvaluateSystem
VAR
    i : INT;
END_VAR




eval.bAllModulesOff := TRUE;
eval.bAnyModuleActive := FALSE;
eval.bAnyModuleFault := FALSE;
eval.bGridOk := TRUE;
eval.rTotalAvailableCurrent := 0;
eval.rMaxTemperature := 0;
eval.iHealthyModules := 0;

get.Events.b_ACPhaselossFault	:=	FALSE;
get.Events.b_ACUndervoltage		:=	FALSE;
get.Events.b_ACOvervoltage		:=	FALSE;


FOR i := 0 TO TO_INT(st_params.ui_NrOfInstalledModules - 1) DO

    IF NOT stData.stModuleData[i].stStatus.bDcSideOff AND stData.stModuleData[i].stStatus.bSlowStartup THEN
        eval.bAllModulesOff := FALSE;
        eval.bAnyModuleActive := TRUE;
        eval.iHealthyModules := eval.iHealthyModules + 1;
    END_IF

    (* Sum current *)
    eval.rTotalAvailableCurrent := eval.rTotalAvailableCurrent +
        stData.stModuleData[i].ravilableCurrentDc;

    (* Max temp *)
    IF stData.stModuleData[i].rTemprature > eval.rMaxTemperature THEN
        eval.rMaxTemperature := stData.stModuleData[i].rTemprature;
    END_IF

    (* Fault detection *)
    IF stData.stModuleData[i].stStatus.bModuleError OR
       stData.stModuleData[i].stStatus.bOutputShortCircuit OR
       stData.stModuleData[i].stStatus.bOutputOverVoltage THEN
        eval.bAnyModuleFault := TRUE;
    END_IF

    (* Grid check *)
    IF stData.stModuleData[i].stStatus.bPhaseLost THEN
		get.Events.b_ACPhaselossFault := TRUE;
		eval.bGridOk := FALSE;
	END_IF

   	IF stData.stModuleData[i].stStatus.bInputOverVoltage THEN
		get.Events.B_ACOvervoltage := TRUE;
		eval.bGridOk := FALSE;
	END_IF
	
	IF stData.stModuleData[i].stStatus.bInputUnderVoltage THEN
		get.Events.B_ACUndervoltage := TRUE;
		eval.bGridOk := FALSE;
    END_IF

END_FOR
END_METHOD

METHOD GetDiagnostics 
VAR_IN_OUT
	AddError		: ARRAY [*] OF FB_AddErrorST;
	a_ActiveEvents	: ARRAY [*] OF ST_ErrorStruct;
	w_Index			: WORD;
END_VAR

(*Module Output OverVoltage Alarm*)	AddError[w_Index](
		b_ErrorTrig			:= st_params.b_ACDCChargerFitted AND (BuscouplerState <> 8),
		out_ST_Error		:= a_ActiveEvents[w_Index],
		w_ErrorID			:= 1,
		e_ObjectID			:= e_ID,
		s_Message			:= 'Buscoupler not found',
		e_sev				:= eseverity.Warning,
		t_TriggerTime		:= T#2S
);
w_Index := w_Index +1;

(*Module Output OverVoltage Alarm*)	AddError[w_Index](
		b_ErrorTrig			:= get.Events.B_ACPhaselossFault,
		out_ST_Error		:= a_ActiveEvents[w_Index],
		w_ErrorID			:= 2,
		e_ObjectID			:= e_ID,
		s_Message			:= 'Input phase missing',
		e_sev				:= eseverity.Warning,
		t_TriggerTime		:= T#1S
);
w_Index := w_Index +1;

(*Module Output OverVoltage Alarm*)	AddError[w_Index](
		b_ErrorTrig			:= get.Events.B_ACOvervoltage,
		out_ST_Error		:= a_ActiveEvents[w_Index],
		w_ErrorID			:= 3,
		e_ObjectID			:= e_ID,
		s_Message			:= 'Input Overvoltage detected',
		e_sev				:= eseverity.Warning,
		t_TriggerTime		:= T#1S
);
w_Index := w_Index +1;

(*Module Output OverVoltage Alarm*)	AddError[w_Index](
		b_ErrorTrig			:= get.Events.B_ACUndervoltage,
		out_ST_Error		:= a_ActiveEvents[w_Index],
		w_ErrorID			:= 4,
		e_ObjectID			:= e_ID,
		s_Message			:= 'Input Undervoltage detected',
		e_sev				:= eseverity.Warning,
		t_TriggerTime		:= T#1S
);
w_Index := w_Index +1;

(*Module Output OverVoltage Alarm*)	AddError[w_Index](
		b_ErrorTrig			:= get.Events.b_FailedToGenerateDCOutput,
		out_ST_Error		:= a_ActiveEvents[w_Index],
		w_ErrorID			:= 5,
		e_ObjectID			:= e_ID,
		s_Message			:= 'Charger failed to generate output',
		e_sev				:= eseverity.Warning,
		t_TriggerTime		:= T#1S
);





















(*
(*Module Output OverVoltage Alarm*)	AddError[w_Index](
		b_ErrorTrig			:= diag.bError_OutputOV,
		out_ST_Error		:= a_ActiveEvents[w_Index],
		w_ErrorID			:= 13,
		e_ObjectID			:= eObject_ID.NeutralTransformer,
		s_Message			:= 'module output overvoltage alarm',
		e_sev				:= eseverity.Normalshutdown,
		t_TriggerTime		:= T#2S
);
w_Index := w_Index +1;

(*Module OverTemp Alarm*)	AddError[w_Index](
		b_ErrorTrig			:= diag.bError_OverTemp,
		out_ST_Error		:= a_ActiveEvents[w_Index],
		w_ErrorID			:= 14,
		s_Message			:= 'module overtemperature alarm',
		e_sev				:= eseverity.Normalshutdown,
		t_TriggerTime		:= T#2S
);
w_Index := w_Index +1;

(*Short Circuit Alarm*)	AddError[w_Index](
		b_ErrorTrig			:= diag.bError_ShortCircuit,
		out_ST_Error		:= a_ActiveEvents[w_Index],
		w_ErrorID			:= 15,
		s_Message			:= 'output short circuit alarm',
		e_sev				:= eseverity.Normalshutdown,
		t_TriggerTime		:= T#1S
);
w_Index := w_Index +1;

(*Module Error Alarm*)	AddError[w_Index](
		b_ErrorTrig			:= diag.bError_ModuleError,
		out_ST_Error		:= a_ActiveEvents[w_Index],
		w_ErrorID			:= 16,
		s_Message			:= 'module error/protection alarm',
		e_sev				:= eseverity.Normalshutdown,
		t_TriggerTime		:= T#1S
);
w_Index := w_Index +1;

(*Communication Lost Alarm*)	AddError[w_Index](
		b_ErrorTrig			:= diag.bError_CommLost,
		out_ST_Error		:= a_ActiveEvents[w_Index],
		w_ErrorID			:= 17,
		s_Message			:= 'communication lost alarm',
		e_sev				:= eseverity.Normalshutdown,
		t_TriggerTime		:= T#3S
);
w_Index := w_Index +1;

(*Phase Lost Alarm*)	AddError[w_Index](
		b_ErrorTrig			:= diag.bError_PhaseLost,
		out_ST_Error		:= a_ActiveEvents[w_Index],
		w_ErrorID			:= 18,
		s_Message			:= 'phase lost alarm',
		e_sev				:= eseverity.Normalshutdown,
		t_TriggerTime		:= T#2S
);
w_Index := w_Index +1;


(* ===== WARNINGS ===== *)

(*Input OverVoltage Warning*)	AddError[w_Index](
		b_ErrorTrig			:= diag.bWarn_InputOV,
		out_ST_Error		:= a_ActiveEvents[w_Index],
		w_ErrorID			:= 19,
		s_Message			:= 'input overvoltage warning',
		e_sev				:= eseverity.Warning,
		b_AutoClear			:= TRUE
);
w_Index := w_Index +1;

(*Input UnderVoltage Warning*)	AddError[w_Index](
		b_ErrorTrig			:= diag.bWarn_InputUV,
		out_ST_Error		:= a_ActiveEvents[w_Index],
		w_ErrorID			:= 20,
		s_Message			:= 'input undervoltage warning',
		e_sev				:= eseverity.Warning,
		b_AutoClear			:= TRUE
);
w_Index := w_Index +1;

(*Fan Error Warning*)	AddError[w_Index](
		b_ErrorTrig			:= diag.bWarn_FanError,
		out_ST_Error		:= a_ActiveEvents[w_Index],
		w_ErrorID			:= 21,
		s_Message			:= 'fan error warning',
		e_sev				:= eseverity.Warning,
		b_AutoClear			:= TRUE
);
w_Index := w_Index +1;

(*Power Limitation Warning*)	AddError[w_Index](
		b_ErrorTrig			:= diag.bWarn_PowerLimit,
		out_ST_Error		:= a_ActiveEvents[w_Index],
		w_ErrorID			:= 22,
		s_Message			:= 'power limitation warning',
		e_sev				:= eseverity.Warning,
		b_AutoClear			:= TRUE
);
w_Index := w_Index +1;

(*Temperature High Warning*)	AddError[w_Index](
		b_ErrorTrig			:= diag.bWarn_TempHigh,
		out_ST_Error		:= a_ActiveEvents[w_Index],
		w_ErrorID			:= 23,
		s_Message			:= 'module temperature high warning',
		e_sev				:= eseverity.Warning,
		b_AutoClear			:= TRUE
);
w_Index := w_Index +1;

*)
END_METHOD

METHOD PRIVATE HandleCanCommunication
VAR
    i, j : INT;
END_VAR





//POLLING (requestin to read data)
IF TxQueue.TxCounter = RxQueue.TxCounter AND NumberOfMessagesToSend > 0 THEN

    CASE Step OF
        0: TxQueue.TxMessages[txIndex].cobId := BuildCanId(16#01, GroupID);
        1: TxQueue.TxMessages[txIndex].cobId := BuildCanId(16#02, GroupID);
        2: TxQueue.TxMessages[txIndex].cobId := BuildCanId(16#04, GroupID);
        3: TxQueue.TxMessages[txIndex].cobId := BuildCanId(16#06, GroupID);
        4: TxQueue.TxMessages[txIndex].cobId := BuildCanId(16#0C, GroupID);
    END_CASE

    TxQueue.TxMessages[txIndex].length := 8;

    FOR j := 0 TO 7 DO
        TxQueue.TxMessages[txIndex].data[j] := 0;
    END_FOR

    txIndex := txIndex + 1;
    IF txIndex > 4 THEN txIndex := 0; END_IF

    Step := Step + 1;
    IF Step > 4 THEN Step := 0; END_IF

END_IF


//COMMANDS 
CASE get.e_SystemStatus OF

    //MODULE OFF Command
	eACDCChargerState.stopping,  eACDCChargerState.fault:
        TxQueue.TxMessages[5].cobId := BuildCanId(16#1A, GroupID);
        TxQueue.TxMessages[5].data[0] := 1;
        TxQueue.TxMessages[5].length := 8;


    // MODULE ON Command
    eACDCChargerState.starting,  eACDCChargerState.running:
        TxQueue.TxMessages[5].cobId := BuildCanId(16#1A, GroupID);
        TxQueue.TxMessages[5].data[0] := 0;
        TxQueue.TxMessages[5].length := 8;

END_CASE


//SETPOINT CMD 
IF get.e_SystemStatus = eACDCChargerState.starting OR get.e_SystemStatus = eACDCChargerState.running THEN

    voltage_mV := REAL_TO_UDINT(rChargerVoltageSetpoint * 1000);
    current_mA := REAL_TO_UDINT(rChargerCurrentSetpoint * 1000);

    TxQueue.TxMessages[6].cobId := BuildCanId(16#1C, GroupID);

    TxQueue.TxMessages[6].data[0] := TO_BYTE(SHR(voltage_mV,24));
    TxQueue.TxMessages[6].data[1] := TO_BYTE(SHR(voltage_mV,16));
    TxQueue.TxMessages[6].data[2] := TO_BYTE(SHR(voltage_mV,8));
    TxQueue.TxMessages[6].data[3] := TO_BYTE(voltage_mV);

    TxQueue.TxMessages[6].data[4] := TO_BYTE(SHR(current_mA,24));
    TxQueue.TxMessages[6].data[5] := TO_BYTE(SHR(current_mA,16));
    TxQueue.TxMessages[6].data[6] := TO_BYTE(SHR(current_mA,8));
    TxQueue.TxMessages[6].data[7] := TO_BYTE(current_mA);

    TxQueue.TxMessages[6].length := 8;

END_IF


//TX TRIGGER 
TxQueue.NoOfTxMessages := TO_UINT(NumberOfMessagesToSend);
TxQueue.TxCounter := TxQueue.TxCounter + 1;
END_METHOD

METHOD limitation : REAL
VAR_INPUT
END_VAR

VAR_INST
	rAvailableChargePower 		: REAL;
	rRampUp			: REAL;
	rRampDown		: REAL;	
END_VAR
limitation := r_MaxChargeCurrent + r_SystemCurrent + stData.rSystemOutCurrentDc;

//// ramp
//rRampUp   := 0.5;   // slow increase
//rRampDown := 5.0;   // fast decrease

//IF stData.rSystemOutCurrentDc > rAvailableChargePower THEN
//    // reduce fast 
//    rMaxLimit := MAX(stData.rSystemOutCurrentDc - rRampDown, rAvailableChargePower);
//ELSE
//    // increase slowly (avoid jump)
//    rMaxLimit := MIN(stData.rSystemOutCurrentDc + rRampUp, rAvailableChargePower);
//END_IF;

//get.Events.b_BatteryLimitDeratingActive := bms.r_MaxChargeCurrentAllowed + bms.r_SystemCurrent
END_METHOD

METHOD MapStatusToStruct : ST_ModuleStatus
VAR_INPUT
    Status2 : BYTE;   // Received status byte 2
    Status1 : BYTE;   // Received status byte 1
    Status0 : BYTE;   // Received status byte 0
END_VAR
VAR
    result : ST_ModuleStatus;
END_VAR



(* ------------------- STATUS 2 ------------------- *)
result.bPfcOff            := (Status2 AND 16#80) <> 0;  // Bit 7
result.bInputOverVoltage  := (Status2 AND 16#40) <> 0;  // Bit 6
result.bInputUnderVoltage := (Status2 AND 16#20) <> 0;  // Bit 5
result.bInputAsymmetry    := (Status2 AND 16#10) <> 0;  // Bit 4
result.bPhaseLost         := (Status2 AND 16#08) <> 0;  // Bit 3
result.bLoadSharingError  := (Status2 AND 16#04) <> 0;  // Bit 2
result.bModuleIdDuplicate := (Status2 AND 16#02) <> 0;  // Bit 1
result.bPowerLimitation   := (Status2 AND 16#01) <> 0;  // Bit 0

(* ------------------- STATUS 1 ------------------- *)
result.bCanTimeout        := (Status1 AND 16#80) <> 0;  // Bit 7
result.bSlowStartup       := (Status1 AND 16#40) <> 0;  // Bit 6
result.bOutputOverVoltage := (Status1 AND 16#20) <> 0;  // Bit 5
result.bTempHigh          := (Status1 AND 16#10) <> 0;  // Bit 4
result.bFanError          := (Status1 AND 16#08) <> 0;  // Bit 3
result.bModuleProtection  := (Status1 AND 16#04) <> 0;  // Bit 2
result.bModuleError       := (Status1 AND 16#02) <> 0;  // Bit 1
result.bDcSideOff         := (Status1 AND 16#01) <> 0;  // Bit 0

(* ------------------- STATUS 0 ------------------- *)
result.bDischargeAbnormal  := (Status0 AND 16#20) <> 0; // Bit 5
result.bMpptSwitchMode     := (Status0 AND 16#10) <> 0; // Bit 4
result.bPfcAbnormal        := (Status0 AND 16#08) <> 0; // Bit 3
result.bInternalCommError  := (Status0 AND 16#04) <> 0; // Bit 2
result.bOutputShortCircuit := (Status0 AND 16#01) <> 0; // Bit 0

MapStatusToStruct := result;  // return struct
END_METHOD

METHOD ReadingRx : BOOL
VAR_INPUT
END_VAR
VAR_INST
	rxID : UDINT;                      // received CAN identifier
	commandNo : UDINT;                  // decoded command number
    deviceNo : UDINT;                   // decoded device number
    errorCode : UDINT;                  // decoded error code
	ModuleAddr : BYTE;
    ControllerAddr : BYTE;
	rxData : ARRAY[0..7] OF USINT;      // received data buffer
	tmpFloat : ARRAY[0..3] OF BYTE;
END_VAR
VAR_INST
	mydword : DWORD;
	mydword2 : DWORD;
    iWd         : INT;
    rxIndex     : INT;

    tModuleWd   : ARRAY [0..10] OF TON;
    bKickModule : ARRAY [0..10] OF BOOL;;
	stEmptyModule : ST_ModuleData; // all fields = 0 by default
	
	TempVoltage : ARRAY[0..2] OF REAL;
	Divider	:	UINT;
END_VAR



// Reset kick flags every cycle
FOR iWd := 0 TO 10 DO
    bKickModule[iWd] := FALSE;
END_FOR


// Receive and decode data
IF RxQueue.RxCounter <> TxQueue.RxCounter THEN
	b_ModuleCommunicationLost := FALSE;
    FOR rxIndex := 0 TO TO_INT(MAX(0, RxQueue.NoOfRxMessages - 1)) DO//max(0,NumberOfMessagesToSend-1) DO

        rxID := RxQueue.RxMessages[rxIndex].cobId AND 16#1FFFFFFF;;     // read CAN identifier
        rxData := RxQueue.RxMessages[rxIndex].Data;  // copy payload
		
		//// extract command from COB-ID  cmd := TO_BYTE(SHR(msg.cobId,16) AND 16#3F);

        (* decode identifier fields according to GCP protocol *)
        errorCode := TO_BYTE(SHR(rxID , 26) AND 16#7);       // bits 28-26
        deviceNo  := TO_BYTE(SHR(rxID , 22) AND 16#F);       // bits 25-22
        commandNo := TO_BYTE(SHR(rxID , 16) AND 16#3F);      // bits 21-16
     //   ModuleAddr     := TO_BYTE(SHR(rxID , 8)  AND 16#FF); // bits 15-8 (source address)
	//	ControllerAddr := TO_BYTE(rxID AND 16#FF);           // bits 7-0  (target address)
	    ControllerAddr     := TO_BYTE(SHR(rxID , 8)  AND 16#FF); 
		ModuleAddr := TO_BYTE(rxID AND 16#FF);          


        CASE commandNo OF

        (* ---- response: system/group voltage & current (float) ---- *)
       1:// 16#01:
            tmpFloat[0] := rxData[0];
            tmpFloat[1] := rxData[1];
            tmpFloat[2] := rxData[2];
            tmpFloat[3] := rxData[3];
			
			
			//SHL(TO_DWORD(readData[i-1]), 16) OR TO_DWORD(readData[i]);
			mydword := SHL(TO_DWORD(tmpFloat[0]), 24) OR SHL(TO_DWORD(tmpFloat[1]), 16) OR SHL(TO_DWORD(tmpFloat[2]), 8) OR TO_DWORD(tmpFloat[3]);
			
            MEMCPY(ADR(stData.rSystemOutVoltageDc), ADR(mydword), 4);  // copy bytes into REAL

            tmpFloat[0] := rxData[4];
            tmpFloat[1] := rxData[5];
            tmpFloat[2] := rxData[6];
            tmpFloat[3] := rxData[7];
			
			mydword2 := SHL(TO_DWORD(tmpFloat[0]), 24) OR SHL(TO_DWORD(tmpFloat[1]), 16) OR SHL(TO_DWORD(tmpFloat[2]), 8) OR TO_DWORD(tmpFloat[3]);
			
            MEMCPY(ADR(stData.rSystemOutCurrentDc), ADR(mydword2), 4);

        (* ---- response: module count ---- *)
      2://  16#02:
            stData.rNumberOfModules := rxData[2];                     // number of modules
			
	3://	16#03: 
			bKickModule[ModuleAddr] := TRUE;
       			 // convert big-endian float to REAL
			tmpFloat[0] := rxData[3];
			tmpFloat[1] := rxData[2];
			tmpFloat[2] := rxData[1];
			tmpFloat[3] := rxData[0];
			MEMCPY(ADR(stData.stModuleData[ModuleAddr].rOutVoltageDc), ADR(tmpFloat), 4); // per-module output voltage
	
			tmpFloat[0] := rxData[7];
			tmpFloat[1] := rxData[6];
			tmpFloat[2] := rxData[5];
			tmpFloat[3] := rxData[4];
			MEMCPY(ADR(stData.stModuleData[ModuleAddr].rOutCurrentDc), ADR(tmpFloat), 4); // per-module output current
				
			
	4: //	16#04:  // module status
			bKickModule[ModuleAddr] := TRUE;
			
            stData.stModuleData[ModuleAddr].rTemprature := TO_SINT(rxData[4]);
            stData.stModuleData[ModuleAddr].rStatus2   	:= rxData[5];
            stData.stModuleData[ModuleAddr].rStatus1    := rxData[6];
            stData.stModuleData[ModuleAddr].rStatus0    := rxData[7];
			(* decode bits into struct *)
			stData.stModuleData[ModuleAddr].stStatus :=	MapStatusToStruct(Status2 := rxData[5], Status1 := rxData[6], Status0 := rxData[7]);

     6://   16#06:  // AC input voltage
	 		bKickModule[ModuleAddr] := TRUE;
			
    		stData.stModuleData[ModuleAddr].rVoltageL1L2 := TO_REAL(rxData[0]*256 + rxData[1]) * 0.1;
            stData.stModuleData[ModuleAddr].rVoltageL2L3 := TO_REAL(rxData[2]*256 + rxData[3]) * 0.1;
            stData.stModuleData[ModuleAddr].rVoltageL3L1 := TO_REAL(rxData[4]*256 + rxData[5]) * 0.1;

   12://     16#0C:  // external voltage / available current
   			bKickModule[ModuleAddr] := TRUE;
			
        	stData.stModuleData[ModuleAddr].rExternalVoltageDc  := TO_REAL(rxData[0]*256 + rxData[1]) * 0.1;
            stData.stModuleData[ModuleAddr].ravilableCurrentDc 	:= TO_REAL(rxData[2]*256 + rxData[3]) * 0.1;


        END_CASE

    END_FOR	

	TxQueue.RxCounter := RxQueue.RxCounter;

	tComWatchdog(IN := FALSE);
ELSE
		
	(* Communication *)
	tComWatchdog(IN := TRUE AND NOT bResetFault, PT := T#10S);
	IF tComWatchdog.Q THEN
		stData.rNumberOfModules := 0;
		stData.rSystemOutCurrentDc := 0;
		stData.rSystemOutVoltageDc :=0;
		b_ModuleCommunicationLost := TRUE;
	END_IF

END_IF




// watchdog 
FOR iWd := 0 TO 10 DO

    // Restart watchdog if message received
    IF bKickModule[iWd] THEN
        tModuleWd[iWd](IN := FALSE);
    END_IF

    // Run watchdog
    tModuleWd[iWd](IN := TRUE, PT := T#5S);

    // Timeout handling
    IF tModuleWd[iWd].Q THEN
        stData.stModuleData[iWd] := stEmptyModule;   // reset 
        stData.stModuleData[iWd].bValid := FALSE;
    ELSE
        stData.stModuleData[iWd].bValid := TRUE;
    END_IF
	
	// to prevent jump in current set
	IF (NOT bValidPrev[iWd]) AND stData.stModuleData[iWd].bValid THEN
    	bFreezeCurrent := TRUE;
	END_IF

	bValidPrev[iWd] := stData.stModuleData[iWd].bValid;
	
	
END_FOR

Divider := 0;
TempVoltage[0] := 0;
TempVoltage[1] := 0;
TempVoltage[2] := 0;

FOR iWd := 0 TO 10 DO
	IF stdata.stModuleData[iWd].bValid THEN
		TempVoltage[0] := TempVoltage[0] + stData.stModuleData[iWd].rVoltageL1L2;
		TempVoltage[1] := TempVoltage[1] + stData.stModuleData[iWd].rVoltageL2L3;
		TempVoltage[2] := TempVoltage[2] + stData.stModuleData[iWd].rVoltageL3L1;
		Divider := Divider +1;
	END_IF
END_FOR

get.ar_ACvoltage[Phases.L1] := TempVoltage[0]/MAX(divider,1);
get.ar_ACvoltage[Phases.L2] := TempVoltage[1]/MAX(divider,1);
get.ar_ACvoltage[Phases.L3] := TempVoltage[2]/MAX(divider,1);
get.ar_ACvoltage[Phases.AVG] := ((get.ar_ACvoltage[Phases.L1] + get.ar_ACvoltage[Phases.L2] + get.ar_ACvoltage[Phases.L3]) / 3 );

get.r_DcCurrent := stdata.rSystemOutCurrentDc;
get.r_DcVoltage := stdata.rSystemOutVoltageDc;
get.r_DcPower 	:= (stdata.rSystemOutCurrentDc * stdata.rSystemOutVoltageDc)/1000;

get.ACmeasurements.ar_ActivePower[0] := get.r_DcPower/0.95;
IF get.ar_ACvoltage[Phases.AVG] > 0 THEN
	get.ACmeasurements.ar_Current[0] := (1000*get.r_DcPower/0.95)/get.ar_ACvoltage[Phases.AVG]/1.73;
ELSE
	get.ACmeasurements.ar_Current[0] := 0;
END_IF
get.r_AvailablePower := (stdata.stModuleData[0].ravilableCurrentDc * stdata.stModuleData[0].rExternalVoltageDc) + 
						(stdata.stModuleData[1].ravilableCurrentDc * stdata.stModuleData[1].rExternalVoltageDc);


//IF diag.bError_PhaseLost
//get.Events.b_ACPhaseLossError := diag.bError_PhaseLost;
END_METHOD

METHOD Reset : BOOL

IF get.e_SystemStatus = eACDCChargerState.Fault THEN
	get.e_SystemStatus := eACDCChargerState.init;
	get.Events.b_FailedToGenerateDCOutput := FALSE;
END_IF

Reset := TRUE;
(*
io.b_ResetOverCurrentProtection := get.events.b_OvercurrentAlarm;
Reset := NOT get.events.b_OvercurrentAlarm;
*)
END_METHOD

METHOD PRIVATE RunStateMachine
VAR_INPUT
END_VAR





IF b_ModuleCommunicationLost AND  get.e_SystemStatus <> eACDCChargerState.fault THEN
    get.e_SystemStatus := eAcDcChargerState.off;
END_IF

CASE get.e_SystemStatus OF

	eACDCChargerState.off:
		IPSRequest.b_Demand_HVDC := false;
	 	IF NOT b_ModuleCommunicationLost THEN
			get.e_SystemStatus := eACDCChargerState.Standby;
		END_IF
	
	eACDCChargerState.Standby:
		IPSRequest.b_Demand_HVDC := false;
		IF set.b_Enable AND NOT get.events.b_SOCLimitReached AND eval.bGridOK THEN
			IPSRequest.b_Demand_HVDC := true;
			if main_fast.InternalPowerSupply.Get.b_HVDCAvailable then
				get.e_SystemStatus := eACDCChargerState.starting;
			end_if
		END_IF
	
	eACDCChargerState.starting:	
		IF NOT eval.bAllModulesOff THEN    // at least one module is on
			get.e_SystemStatus := eACDCChargerState.running;
		END_IF
		
	eACDCChargerState.running:	
		IF NOT set.b_Enable OR get.events.b_SOCLimitReached OR NOT eval.bGridOK THEN 
			get.e_SystemStatus := eACDCChargerState.stopping;
		END_IF
	
	eACDCChargerState.stopping:	
		IF eval.bAllModulesOff THEN
			get.e_SystemStatus := eACDCChargerState.Standby;
		END_IF
END_CASE
END_METHOD

METHOD PRIVATE SafetyCheck
VAR_INPUT
END_VAR


 


(* Window check *)
bVoltageWindowOk := stData.rSystemOutVoltageDc > r_SystemVoltage - 5.0;
tCheck(in:= NOT eval.bAllModulesOff AND not bVoltageWindowOk, PT := T#5S);

IF tCheck.Q THEN
	get.Events.b_FailedToGenerateDCOutput := TRUE;
	get.e_SystemStatus := eACDCChargerstate.fault;
END_IF
END_METHOD

METHOD PRIVATE UpdateStData
VAR
    i : INT;
END_VAR
VAR_INST
	stDataLast : ST_Data;
END_VAR




// Loop through modules
FOR i := 0 TO TO_INT(stData.rNumberOfModules) DO
    IF stData.stModuleData[i].stStatus.bCanTimeout THEN
        // Keep previous good value
        stData.stModuleData[i] := stDataLast.stModuleData[i];
    ELSE
        // Save new value as last known good
        stDataLast.stModuleData[i] := stData.stModuleData[i];
    END_IF
END_FOR

// Save system-level values
IF NOT b_ModuleCommunicationLost THEN
    stDataLast.rSystemOutVoltageDc := stData.rSystemOutVoltageDc;
    stDataLast.rSystemOutCurrentDc := stData.rSystemOutCurrentDc;
    stDataLast.rNumberOfModules   := stData.rNumberOfModules;
END_IF
END_METHOD

METHOD PRIVATE ValidateOutput
VAR_INPUT
END_VAR




IF get.e_SystemStatus = eACDCChargerstate.running THEN

    IF ABS(stData.rSystemOutVoltageDc - rChargerVoltageSetpoint) > rChargerVoltageSetpoint * 0.1 THEN
        bWarning := TRUE;
    END_IF

    IF ABS(stData.rSystemOutCurrentDc - rChargerCurrentSetpoint) > rChargerCurrentSetpoint * 0.2 THEN
        bWarning := TRUE;
    END_IF
ELSE
	bWarning := FALSE;	
END_IF
END_METHOD

END_FUNCTION_BLOCK

// ---- POUs/Objects/DCLink/FB_DCLink.TcPOU
FUNCTION_BLOCK FB_DCLink
VAR_IN_OUT CONSTANT
	st_params					: ST_DCLink_params;
END_VAR

VAR_INPUT
	r_InvCurrentDC				: REAL;	
	r_BattCurrent				: REAL;
	r_DCbusVoltage				: REAL;	
	r_BattCCL					: REAL;
	r_BattDCL					: REAL;
	b_DCsafetyOK				: BOOL;
	set							: ST_DCLink_set;
END_VAR

VAR_OUTPUT
	get						: ST_DCLink_Get;
	b_DcEDM 		 		: BOOL;
	st_PowerDemand			: ST_InternalPowerSupply_PowerDemand;
END_VAR

VAR
	TempEDMForce			:	BOOL;
	IO 						: FB_CNV520;
	//Powermeter				: fb_shuntbournsSSD;
	RS_DCBusEnableReq			: RS;
	r_trigEnableBus			:	R_trig;
END_VAR

VAR CONSTANT
	e_ID 				: eObject_ID := eObject_ID.DC_Switchgear;
END_VAR

//Get power data
//PowerMeter(IP := st_params.IP,
//			b_enable := settings.Configuration.b_DCbuscoupling,
//			UpdateInterval := T#500MS);

IO(
	b_enable				:= settings.Configuration.b_DCbuscoupling,				
	UpdateInterval			:= T#500MS,
	DigitalOutput_Enable	:= RS_DCBusEnableReq.Q1 AND (main_fast.InternalPowerSupply.Get.b_HVDCAvailable OR st_params.AllowClosingOnDeadBus),
	st_params := st_params
);

st_PowerDemand.b_Demand_HVDC := RS_DCBusEnableReq.Q1;
r_trigEnableBus(clk := set.b_DCBusEnable);

RS_DCBusEnableReq(	SET := r_trigEnableBus.Q AND NOT IO.CommFault,
				RESET1 := NOT set.b_DCBusEnable 
							OR NOT b_DCsafetyOK 
							OR get.events.OvercurrentTrip);

//get.events.OvervoltageNOK := powermeter.events.b_OvervoltageError;
get.b_DCCouplingState := io.DigitalInput2;
b_DcEDM := NOT io.DigitalInput2 OR TempEDMForce;
get.Powerdata REF= IO.Powerdata;

PowerLimitControl(
	Voltage			:= r_DCbusvoltage,
	DCC_current 	:= get.Powerdata.Current,
	Inv_Current 	:= r_InvCurrentDC,
	Batt_Current 	:= r_BattCurrent,
	Batt_CCL		:= ABS(r_BattCCL),
	Batt_DCL		:= ABS(r_BattDCL),
	PowerRampRate	:= set.r_PowerRampRate,
	Inv_CPL			=> get.r_BattChargePowerLimit,
	Inv_DPL			=> get.r_BattDischargePowerLimit,
	DCC_CPL			=> get.r_ImportPowerLimit,
	DCC_DPL			=> get.r_ExportPowerLimit,
	DCC_CCL			=> get.r_ImportCurrentLimit,
	DCC_DCL			=> get.r_ExportCurrentLimit);

//Overcurrent protection
OvercurrentProtection(
	get.powerdata.Current, 
	get.r_ImportCurrentLimit, 
	get.r_exportCurrentLimit);

METHOD GetDiagnostics : BOOL
VAR_IN_OUT
	AddError		: ARRAY [*] OF FB_AddErrorST;
	a_ActiveEvents	: ARRAY [*] OF ST_ErrorStruct;
	w_Index			: WORD;
END_VAR

(*Overcurrent trip*)		AddError[w_Index](
		b_ErrorTrig				:= get.Events.OvercurrentTrip,
		out_ST_Error			:= a_ActiveEvents[w_Index],
		w_ErrorID				:= 1,
		e_ObjectID				:= e_id,						//only first call set object ID.
		s_Message				:= 'coupling overcurrent trip',
		e_sev					:= eSeverity.warning,	//<-- maybe normal shutdown?
		b_AutoClear				:= FALSE
		);
	w_Index := w_Index +1;
		
(*Overvoltage  NOK*)		AddError[w_Index](
		b_ErrorTrig				:= get.Events.OvervoltageNOK,
		out_ST_Error			:= a_ActiveEvents[w_Index],
		w_ErrorID				:= 2,
		e_ObjectID				:= e_id,						//only first call set object ID.
		s_Message				:= 'Overvoltage protection not OK',
		e_sev					:= eSeverity.warning,	//<-- maybe normal shutdown?
		b_AutoClear				:= FALSE
		);
	w_Index := w_Index +1;

(*Overvoltage  NOK*)		AddError[w_Index](
		b_ErrorTrig				:= IO.DigitalInput1,
		out_ST_Error			:= a_ActiveEvents[w_Index],
		w_ErrorID				:= 3,
		e_ObjectID				:= e_id,						//only first call set object ID.
		s_Message				:= 'DC surge protection failed',
		e_sev					:= eSeverity.warning,	//<-- maybe normal shutdown?
		b_AutoClear				:= TRUE
		);
	w_Index := w_Index +1;

(*Overvoltage  NOK*)		AddError[w_Index](
		b_ErrorTrig				:= IO.CommFault,
		out_ST_Error			:= a_ActiveEvents[w_Index],
		w_ErrorID				:= 4,
		e_ObjectID				:= e_id,						//only first call set object ID.
		s_Message				:= 'DC IO communication fault',
		e_sev					:= eSeverity.warning,	//<-- maybe normal shutdown?
		b_AutoClear				:= TRUE
		);
	w_Index := w_Index +1;


(*Overvoltage  NOK*)		AddError[w_Index](
		b_ErrorTrig				:= NOT b_DCsafetyOK,
		out_ST_Error			:= a_ActiveEvents[w_Index],
		w_ErrorID				:= 5,
		e_ObjectID				:= e_id,						//only first call set object ID.
		s_Message				:= 'DC safety not ok',
		e_sev					:= eSeverity.warning,	//<-- maybe normal shutdown?
		b_AutoClear				:= TRUE
		);
	w_Index := w_Index +1;	
//(*Overvoltage  NOK*)		AddError[w_Index](
//		b_ErrorTrig				:= Powermeter.CommFault,
//		out_ST_Error			:= a_ActiveEvents[w_Index],
//		w_ErrorID				:= 5,
//		e_ObjectID				:= e_id,						//only first call set object ID.
//		s_Message				:= 'DC powermeter communication fault',
//		e_sev					:= eSeverity.warning,	//<-- maybe normal shutdown?
//		b_AutoClear				:= TRUE
//		);
//	w_Index := w_Index +1;
END_METHOD

METHOD GetWearCounters : BOOL
VAR_INST
	
	MCCBLogger			:	FB_Varlogger;
//	MCCBTripLogger		:	FB_Varlogger;	
END_VAR


MCCBLogger(		TriggerInput := get.b_DCCouplingState, 
						LogItemGroup :=  eLogItemGroupID.DcLink, 
						LogItemName := 'MCCBCnt', 
						LogType := eLogTypes.TrackCycles);
(*
MCCBTripLogger(	TriggerInput := b_MCCBinputShuntTrip, 
						LogItemGroup :=  eLogItemGroupID.DcLink, 
						LogItemName := 'MCCBTripCnt', 
						LogType := eLogTypes.TrackCycles);
*)
						
Wearlogging.SetFloat( eLogItemGroupID.DcLink, 	'Energy', 			eLogTypes.WriteValue, 	REAL_TO_LREAL(get.Powerdata.Energy));
Wearlogging.SetFloat( eLogItemGroupID.DcLink, 	'MaxTempEver', 		eLogTypes.KeepHighestValue, 	REAL_TO_LREAL(get.Powerdata.Temperature));
END_METHOD

METHOD OverCurrentProtection : BOOL
VAR_INPUT
	DCC_Current				: REAL;
	DCC_CCL					: REAL;
	DCC_DCL					: REAL;
END_VAR

VAR_INST
	ton_OCPdelay 			: TON := (PT:= T#2S);
END_VAR
ton_OCPDelay(PT := st_params.OvercurrentTripDelay);

IF RS_DCBusEnableReq.q1 THEN
	IF main_fast.BMS.get.BatteryInfo.e_BMS_PowerOnStatus = ePowerOnStatus.On THEN
		ton_OCPDelay.IN := DCC_current < -DCC_CCL OR DCC_Current > DCC_DCL;
	ELSIF st_params.AllowClosingOnDeadBus THEN
			ton_ocpdelay.IN := DCC_Current < -UINT_TO_INT(st_params.RatedCurrent) OR DCC_Current > st_params.RatedCurrent;
	END_IF
ELSE
	ton_ocpdelay.IN := FALSE;
END_IF
	
IF ton_OCPdelay.Q THEN
	get.events.OvercurrentTrip := TRUE;
END_IF
END_METHOD

METHOD PowerLimitControl : BOOL
VAR_INPUT
	Voltage				: REAL;
	DCC_Current 		: REAL;
	Inv_Current			: REAL;
	Batt_Current		: REAL;
	Batt_CCL			: REAL;
	Batt_DCL			: REAL;
	PowerRampRate		: REAL := 1;
END_VAR


VAR_INST
	Inv_CCL			: REAL;
	Inv_DCL			: REAL;
END_VAR

VAR_OUTPUT
	Inv_CPL			: REAL;
	Inv_DPL			: REAL;
	DCC_CCL 		: REAL;
	DCC_DCL			: REAL;
	DCC_CPL 		: REAL;
	DCC_DPL			: REAL;
	DCC_set			: REAL;
END_VAR
(*
	DC power priority
	auto: 
		- DC power slow ramp, inverter power limited fast through DC power max variable,
			(combination of BMS current max - DC coupling current) 
			>> RESULT: Reduction of battery current causes inverter to immediatly throttle, 
				after which the DC coupling current is reduced with specified ramp.
	inverter: 
		- DC coupling power is reduced first, then inverter is being throttled by batteries directly as usual
			>> CODING: 
				DC coupling current set max = BatteryDischargeLimit - inverter power
				DC coupling current set min = BatteryChargeLimit - inverter power
				Q = LIMIT(DCCS_min, DCCS, DCCS_max);
			
	DCcoupling: 
		- Inverter is reduced first, then DC coupling is throtthled 

	*)
	
CASE set.e_DCpowerPriority OF
	eDCpowerpriority.auto:
	//AUTO mode: inverter first, then bus to maintain battery limits
		//Charge limit of dc coupling
		Inv_CCL := Batt_CCL + DCC_Current; // 500 + (-100) = 400
		IF Inv_current <= -Inv_CCL THEN //Invcurrent < 0 is charging
			DCC_CCL := DCC_CCL - PowerRamprate / 1000;
		ELSIF Inv_current > -Inv_CCL * MAX(0, 1-st_params.DCpowerControlHyst) THEN
			DCC_CCL := DCC_CCL + PowerRamprate / 1000;
		END_IF	
		
		//Discharge limit of dc coupling
		Inv_DCL := Batt_DCL + DCC_Current; // 500 + 100 = 400
		IF Inv_current >= Inv_DCL THEN
			DCC_DCL := DCC_DCL - PowerRamprate / 1000;
		ELSIF Inv_current <= Inv_DCL * MAX(0, 1-st_params.DCpowerControlHyst) THEN
			DCC_DCL := DCC_DCL + PowerRamprate / 1000;
		END_IF	
		
	eDCpowerPriority.DCcoupling:
	//DC coupling priority, will reduce inverter power first
		//Charge limit:
		Inv_CCL := Batt_CCL + DCC_Current;
		Inv_DCL := Batt_DCL + DCC_Current;
		DCC_CCL := Batt_CCL;
		DCC_DCL := Batt_DCL;
		
	eDCpowerpriority.Inverter:
	//Inverter priority, will reduce DC coupling first.	
		DCC_CCL := Batt_CCL + Inv_Current;
		DCC_DCL := Batt_DCL + Inv_Current;
		Inv_CCL := Batt_CCL;
		Inv_DCL := Batt_DCL;	
END_CASE

DCC_DCL := LIMIT(0, DCC_DCL, st_params.RatedCurrent);
DCC_CCL := LIMIT(0, DCC_CCL, st_params.RatedCurrent);

//Power outputs
DCC_DPL := ABS(DCC_DCL * voltage / 1000);
DCC_CPL := ABS(DCC_CCL * voltage / 1000);
Inv_DPL := ABS(Inv_DCL * voltage / 1000);
Inv_CPL := ABS(Inv_CCL * voltage / 1000);
END_METHOD

METHOD Reset : BOOL
VAR_INPUT
END_VAR
get.events.OvercurrentTrip := FALSE;
END_METHOD

END_FUNCTION_BLOCK

// ---- POUs/Objects/DCLink/FB_CNV520.TcPOU
FUNCTION_BLOCK FB_CNV520
VAR_INPUT
	
END_VAR
VAR_OUTPUT
	
END_VAR
VAR
	
	
	WriteOutput			: 	FB_MBWriteSingleReg;
	OutputData			:	WORD;
	StartWriteOutput	:	BOOL;
	OutputWriteError	:	Ton	:=	(PT := T#10S);
	NextStepDelay		:	Ton :=	(PT := T#50MS);
	
	ReadInputs			: 	FB_MBReadRegs;
	DIData				:	ARRAY[0..1] OF WORD;
	StartReadinputs		:	BOOL;	
	InputReadError		:	Ton := (Pt := T#10S);
	
	ReadShuntInputs			: 	FB_MBReadInputRegs;
	ShuntData				:	ARRAY[0..20] OF WORD;
	StartReadShunt			:	BOOL;	
	InputReadShuntError		:	Ton := (Pt := T#10S);
	
	dataInputs				: ARRAY[0..20] OF DWORD;
	lw_Power				: LWORD;  // Unsigned int32
	lw_Energy				: LWORD; // Unsigned int64
	lw_Coulomb				: LWORD; // Signed int64
	
	StartHoldingWrite	:	BOOL;

	TON_UpdateInterval	:	Ton;
	
	State : UINT	:=	0;
	
	AuxSurgeProtectionInput 	AT %I* : BOOL;
	AuxMCCBStateInput 			AT %I* : BOOL;
END_VAR

VAR_INPUT
	b_enable				:	BOOL;

	UpdateInterval			:	TIME 	:=	T#500MS;
	DigitalOutput_Enable	:	BOOL;
END_VAR

VAR_IN_OUT constant
	st_params					: ST_DCLink_params;
END_VAR

VAR_OUTPUT
	AnalogInput			:	REAL;
	DigitalInput1		:	BOOL;
	DigitalInput2		:	BOOL;
	DigitalOutputState	:	BOOL;
	
	Powerdata			:	st_Bourns_powerdata;
	CommFault			:	Bool;
END_VAR


WriteOutput(
	sIPAddr := st_params.IP,
	nTCPPort := 502,
	nUnitID := 247,
	nMBAddr	:=	60,
	nValue := OutputData,
	bExecute := StartWriteOutput,
	tTimeout := T#1000MS
);
OutputWriteError();

Readinputs(
	sIPAddr := ST_params.ip,
	nTCPPort := 502,
	nUnitID := 247,
	nMBAddr	:=	56,
	nQuantity := 1,
	cbLength := SIZEOF(DIData),
	pDestAddr := ADR(DiData),
	bExecute := StartReadinputs,
);
InputReadError();

ReadShuntinputs(
	sIPAddr := st_params.IP,
	nTCPPort := 502,
	nUnitID := 1,
	nMBAddr	:=	0,
	nQuantity := 21,
	cbLength := SIZEOF(ShuntData),
	pDestAddr := ADR(ShuntData),
	bExecute := StartReadshunt,
);
InputReadShuntError();

TON_UpdateInterval(in := NOT TON_UpdateInterval.Q, PT:= UpdateInterval);
NextStepDelay();

CASE State OF
	0:
		IF b_enable AND Ton_UpdateInterval.Q THEN
			State := 10;
		END_IF	
		
	10:
		outputData.0 := DigitalOutput_Enable;
		StartWriteOutput := TRUE;
		state := 11;
		
	11:
		StartWriteOutput := FALSE;
		IF NOT WriteOutput.bBusy THEN
			IF NOT WriteOutput.bError THEN
				DigitalOutputSTate := SEL(outputData.0, FALSE, TRUE);
				OutputWriteError.IN := FALSE;
			ELSE
				OutputWriteError.IN := TRUE;
			END_IF
			NextStepDelay.IN := TRUE;
			
			IF st_params.DIWiredToPLC THEN
				DigitalInput1 := AuxSurgeProtectionInput;
				DigitalInput2 := AuxMCCBStateInput;
				State := 30;
			ELSE
				State := 20;
			END_IF
		END_IF

		
	20:
		IF NextStepDelay.Q THEN
			NextStepDelay.IN := FALSE;
			StartReadInputs := TRUE;
			state := 21;
		END_IF
		
	21:
		StartReadInputs := FALSE;
		IF NOT ReadInputs.bBusy THEN
			IF NOT ReadInputs.bError THEN
				DigitalInput1 := DIData[0].0;
				DigitalInput2 := DIData[0].1;
				AnalogInput := ((WORD_TO_REAL(DIData[1])/4096)+4);
				InputReadError.IN := FALSE;
			ELSE
				InputReadError.IN := TRUE;
			END_IF
			State := 30;
		END_IF
		
	30:
		StartReadShunt := TRUE;
		state := 31;
		
	31:
		StartReadShunt := FALSE;
		IF NOT ReadShuntInputs.bBusy THEN
			IF NOT ReadShuntInputs.bError THEN
				dataInputs[0]	:= SHL(WORD_TO_DWORD(ShuntData[1]), 16) OR (WORD_TO_DWORD(ShuntData[0]));   	
				dataInputs[2]	:= SHL(WORD_TO_DWORD(ShuntData[3]), 16) OR (WORD_TO_DWORD(ShuntData[2])); 		
				dataInputs[4]   := SHL(WORD_TO_DWORD(ShuntData[5]), 16) OR (WORD_TO_DWORD(ShuntData[4]));   
				dataInputs[18]	:= SHL(WORD_TO_DWORD(ShuntData[19]), 16) OR (WORD_TO_DWORD(ShuntData[18]));	
				
				lw_Coulomb 		:= SHL(WORD_TO_LWORD(ShuntData[9]), 48) OR SHL(WORD_TO_LWORD(ShuntData[8]), 32) OR 
									SHL(WORD_TO_DWORD(ShuntData[7]), 16) OR (ShuntData[6]);								
				lw_Power     		:= SHL(WORD_TO_DWORD(ShuntData[11]), 16) OR (WORD_TO_DWORD(ShuntData[10]));   	
				lw_Energy 		:= SHL(WORD_TO_LWORD(ShuntData[15]), 48) OR SHL(WORD_TO_LWORD(ShuntData[14]), 32) OR 
									SHL(WORD_TO_DWORD(ShuntData[13]), 16) OR (ShuntData[12]);							
	
				Powerdata.Current			:= TO_REAL(DWORD_TO_DINT(dataInputs[0]))	/ 1000;  // mA to A
				Powerdata.Temperature		:= TO_REAL(DWORD_TO_DINT(dataInputs[2])) / 10;	// 0.1 °C to °C
				Powerdata.Voltage		   	:= TO_REAL(DWORD_TO_DINT(dataInputs[4])) / 1000; // mV to V
				Powerdata.Power			:= TO_REAL(lw_power) / 10000; // 0.1 W to kW	
				Powerdata.Energy			:= TO_REAL(lw_energy) / 1000;  // Wh to Kwh
				
				InputReadShuntError.IN := FALSE;
			ELSE
				InputReadShuntError.IN := TRUE;
			END_IF
			State := 0;
		END_IF
END_CASE

CommFault := inputReaderror.Q OR outputWriteError.Q OR InputReadShuntError.q;

END_FUNCTION_BLOCK

// ---- POUs/Objects/HartingIO/FB_HartingIO.TcPOU
FUNCTION_BLOCK FB_HartingIO

VAR_IN_OUT CONSTANT
	st_params 			: ST_HartingIO_params;
END_VAR

VAR_INPUT
	set 				: ST_HartingIO_Set;
	SystemOperating		: BOOL;
	SystemEmStop		: BOOL;
END_VAR

VAR_OUTPUT
	Get								:	ST_HartingIO_Get;
	b_SystemRestartTrigger			: 	BOOL;
END_VAR

VAR	
	b_ExtDO1				AT %Q* : BOOL;	
	b_ExtDO2				AT %Q* : BOOL;
	b_ExtDI1				AT %I* : BOOL;
	b_ExtDI2				AT %I* : BOOL;
	i_AO1					AT %Q* : INT;
	i_AO2					AT %Q* : INT;
END_VAR

b_ExtDO1 := configureOutputContact(SignalSelect := st_params.PrimaryOutputContactSignal); 
b_ExtDO2 := configureOutputContact(SignalSelect := st_params.SecondaryOutputContactSignal); 
 
configureInputcontact(SignalSelect := st_params.PrimaryInputContactSignal, b_ExtDI1); 
//configureInputcontact(SignalSelect := st_params.SecondaryInputContactSignal, b_ExtDI2); 
get.b_DigitalInput1Active := b_ExtDi1;
get.b_DigitalInput2Active := b_ExtDi2;

AutoRestartAfterExtEmstop();


CASE st_params.AO1Target OF
	eAOtarget.manual	: i_AO1 := AnalogOutputScaling(set.r_manualAnalogOutput);
	eAOtarget.Genset	: i_AO1 := AnalogOutputScaling(set.r_gensetAnalogOutput);
	eAOtarget.hPU		: i_AO1 := AnalogOutputScaling(set.r_HpuAnalogOutput);
END_CASE

CASE st_params.AO2Target OF
	eAOtarget.manual	: i_AO2 := AnalogOutputScaling(set.r_manualAnalogOutput);
	eAOtarget.Genset	: i_AO2 := AnalogOutputScaling(set.r_gensetAnalogOutput);
	eAOtarget.hPU		: i_AO2 := AnalogOutputScaling(set.r_HpuAnalogOutput);
END_CASE

METHOD AnalogOutputScaling : INT
VAR_INPUT
	IN : REAL;
END_VAR

VAR_INST
	scale_analogOutput			: FB_ctrl_Scale;
	st_paramsScale				: ST_ctrl_scale_params;
END_VAR
//Scale real to analog output
st_paramsScale.fInMax:= 100;
	st_paramsScale.fInMin:= 0;
	st_paramsScale.fOutMax:= 16#8000 -1;
	st_paramsScale.fOutMin:= 0;
	st_paramsScale.tCtrlCycleTime := T#1MS;
	st_paramsScale.tTaskCycleTime := T#1MS;

scale_analogOutput(stParams:= st_paramsScale,
	fIn:= IN);
	AnalogOutputScaling := TO_INT(scale_analogOutput.fOut);
END_METHOD

METHOD AutoRestartAfterExtEmstop : BOOL
VAR_INST
	SystemLastOperation : BOOL;
	
	ExtEmStopRestartTriggered	: BOOL;
	R_TrigoperatingReset		: R_TRIG;
	Ton_DelayCheckState	: TON := (PT:=T#2S);	
END_VAR
IF get.b_ExtEMstopActive THEN
	ExtEmStopRestartTriggered := TRUE;
END_IF

R_TrigoperatingReset(CLK := SystemOperating);
IF R_TrigoperatingReset.Q AND ExtEmStopRestartTriggered THEN
	ExtEmStopRestartTriggered := FALSE;
END_IF

IF NOT SystemEmStop AND SystemOperating THEN
	SystemLastOperation := TRUE;
END_IF

Ton_DelayCheckState(IN := NOT ExtEmStopRestartTriggered AND NOT SystemOperating);
IF ton_DelayCheckState.Q THEN
	SystemLastOperation := FALSE;
END_IF

b_SystemRestartTrigger := SystemLastOperation AND ExtEmStopRestartTriggered;
END_METHOD

METHOD ConfigureInputContact : BOOL
VAR_INPUT
	SignalSelect			: 	eInputSignal;
	InputStatus				:	BOOL;
END_VAR
get.b_GenLowFuel 				:= (SignalSelect = eInputSignal.GenLowFuel) 	AND InputStatus;
get.b_ExtSystemShutdownRequest 	:= (SignalSelect = eInputSignal.StopOperation) 	AND InputStatus;
get.b_ExtEmstopOK 				:= (SignalSelect = eInputSignal.EMstop) 		AND InputStatus;
END_METHOD

METHOD ConfigureOutputContact : BOOL
VAR_INPUT
	SignalSelect			: eOutputContactSignal;
END_VAR
CASE SignalSelect OF
	eOutputContactSignal.GenStartStop 	: ConfigureOutputContact:= set.w_SwitchControlSignals.0;
	eOutputContactSignal.FireAlarm 		: ConfigureOutputContact:= set.w_SwitchControlSignals.1;
	eOutputContactSignal.HPU			: ConfigureOutputContact:= set.w_SwitchControlSignals.2;
	eOutputContactSignal.SystemActive	: ConfigureOutputContact:= set.w_SwitchControlSignals.3;
	eOutputContactSignal.PVenable		: ConfigureOutputContact:= set.w_SwitchControlSignals.4;
	eOutputContactSignal.None, eOutputContactSignal.ManualOpen	
										:	ConfigureOutputContact := FALSE;
	eOutputContactSignal.ManualClose	:	ConfigureOutputContact := TRUE;
END_CASE
END_METHOD

METHOD GetDiagnostics
VAR_IN_OUT
	AddError		: ARRAY [*] OF FB_AddErrorST;
	a_ActiveEvents	: ARRAY [*] OF ST_ErrorStruct;
	w_Index			: WORD;
END_VAR
	(*Shutdown trigger*)		AddError[w_Index](
					b_ErrorTrig				:= get.b_ExtSystemShutdownRequest,
					out_ST_Error			:= a_ActiveEvents[w_Index],
					w_ErrorID				:= 1,
					e_ObjectID				:= eObject_ID.HartingIO,
					s_Message				:= 'External shutdown triggered',
					e_sev					:= eSeverity.NormalShutdown
				);
				w_Index := w_Index +1;
				
		(*EMstop trigger*)		AddError[w_Index](
					b_ErrorTrig				:= ((st_params.PrimaryInputContactSignal = eInputSignal.emstop) OR (st_params.SecondaryInputContactSignal = eInputSignal.emstop)) AND NOT get.b_ExtEMstopOK,
					out_ST_Error			:= a_ActiveEvents[w_Index],
					w_ErrorID				:= 2,
					e_ObjectID				:= eObject_ID.HartingIO,
					s_Message				:= 'External EMstop triggered',
					e_sev					:= eSeverity.QuickShutdown,
					b_Out					=> get.b_ExtEMstopActive
				);
				w_Index := w_Index +1;
END_METHOD

END_FUNCTION_BLOCK

// ---- POUs/Objects/NeutralTransformer/FB_NeutralTransformer.TcPOU
FUNCTION_BLOCK FB_NeutralTransformer
VAR_OUTPUT
	get									: ST_Neutraltransformer_Get;
END_VAR

VAR_IN_OUT CONSTANT
	st_params							: ST_Neutraltransformer_params;
END_VAR

VAR_INPUT
	b_enable						: BOOL;
	r_CurrentN						: REAL; //N
	r_LineVoltage					: REAL;
	r_VoltageUnbalance				: REAL; //%
	b_NetcontactorFb				: BOOL;
END_VAR

VAR					// LOCAL VARIABLES
	IO								: FB_NeutralTransformer_IO;
END_VAR

IF b_enable THEN
	IO();
	CheckCurrents(get.events, st_params, r_CurrentN);
	CheckTemperatures(get.events, st_params, IO.r_TemperaturePhase, get); 
	CheckVoltages(get.events, st_params, r_VoltageUnbalance, b_netcontactorFB := b_NetcontactorFb);
END_IF

get.b_active := b_enable;

METHOD PROTECTED CheckCurrents
VAR_IN_OUT
	events					: ST_Neutraltransformer_events;
END_VAR

VAR_IN_OUT CONSTANT
	st_params			: ST_NeutralTransformer_Params;
	r_CurrentN			: REAL;
END_VAR

VAR
	r_ratedCurrent : REAL;
END_VAR
r_ratedCurrent :=	TO_REAL(st_params.ui_ratedpower) * 1000 / 230;

LimitTrigger(
	r_HighLimit := r_ratedCurrent * st_params.r_OCTripFactor,
	r_HighWarning := r_ratedCurrent,
	b_HighEnable := TRUE,
	r_lowlimit := 0,
	r_lowWarning := 0,
	b_lowEnable := FALSE,
	r_Hysteresis := 10,
	r_in := r_CurrentN,
	b_warning => events.b_NeutralCurrentHigh,
	b_fault => events.b_NeutralCurrentTooHigh
);

get.r_Powerload := r_CurrentN / r_ratedCurrent * 100;
get.r_RatedPower := st_params.ui_ratedpower;
END_METHOD

METHOD PROTECTED CheckTemperatures
VAR_IN_OUT
	events								: ST_NeutralTransformer_events;
END_VAR
VAR_IN_OUT CONSTANT
	st_params							: ST_NeutralTransformer_params;
	r_tempPhase							: ARRAY [1..3] OF REAL;
END_VAR

VAR_IN_OUT
	get									: ST_Neutraltransformer_get;
END_VAR

VAR 
	w_Index								: WORD;
END_VAR
FOR w_Index:=1 TO 3 DO
	LimitTrigger(
		r_HighLimit := st_params.by_TemperatureHighAlarm,
		r_HighWarning := st_params.by_TemperatureHighWarning,
		b_HighEnable := TRUE,
		r_lowlimit := 0,
		r_lowWarning := 0,
		b_lowEnable := FALSE,
		r_Hysteresis := 5,
		r_in := r_TempPhase[w_Index],
		b_warning => events.b_TemperatureHighPhase[w_Index],
		b_fault => events.b_TemperatureHighPhase[w_Index]
	);
END_FOR

get.r_TemperaturePhase[phases.L1] := r_tempphase[phases.L1];
get.r_TemperaturePhase[phases.L2] := r_tempphase[phases.L2];
get.r_TemperaturePhase[phases.L3] := r_tempphase[phases.L3];
get.r_TemperaturePhase[phases.AVG] := r_tempphase[phases.L1] + r_tempphase[phases.L2] + r_tempphase[phases.L3] / 3;
get.r_TemperaturePhase[phases.maximum] := MAX(r_tempphase[phases.L1], r_tempphase[phases.L2], r_tempphase[phases.L3]);
get.r_TemperaturePhase[phases.minimum] := MIN(r_tempphase[phases.L1], r_tempphase[phases.L2], r_tempphase[phases.L3]);
END_METHOD

METHOD PROTECTED CheckVoltages : BOOL
VAR_IN_OUT
	events 				: ST_NeutralTransformer_events;
END_VAR

VAR_IN_OUT CONSTANT
	st_params				: ST_Neutraltransformer_params;
	r_voltageUnbalance		: REAL;
	b_netcontactorFB		: BOOL;
END_VAR

VAR_INST
	b_VoltageOK				: BOOL;
	sr_warning				: SR;
	sr_Alarm				: SR;
END_VAR
b_voltageOK		:= r_LineVoltage >= settings.GridParams.r_GridVoltageMin;
sr_warning(
	SET1 := r_voltageunbalance >= st_params.by_VoltageUnbalanceWarning AND b_voltageOK, 
	RESET := r_voltageunbalance <= st_params.by_VoltageUnbalanceWarning - 2 OR NOT b_netcontactorFB, 
	Q1 => events.b_VoltageUnbalanceHigh
	);

sr_alarm(
	SET1:= r_voltageunbalance >=st_params.by_VoltageUnbalanceAlarm AND b_voltageOK,
	RESET := r_voltageunbalance <= st_params.by_VoltageUnbalanceWarning OR NOT b_netcontactorFB,
	Q1 => events.b_VoltageUnbalanceTooHigh
	);
END_METHOD

METHOD PUBLIC GetDiagnostics
VAR_IN_OUT
	AddError		: ARRAY [*] OF FB_AddErrorST;
	a_ActiveEvents	: ARRAY [*] OF ST_ErrorStruct;
	w_Index			: WORD;
END_VAR
(*Temp L1 Warning*)		AddError[w_Index](
		b_ErrorTrig			:= get.events.b_TemperatureHighPhase[phases.L1],
		out_ST_Error			:= a_ActiveEvents[w_Index],
		w_ErrorID					:= 1,
		e_ObjectID				:= eObject_ID.NeutralTransformer,
		s_Message				:= 'high temperature L1 warning',
		e_sev					:= eseverity.Warning,
		b_AutoClear			:= TRUE
	);
	w_Index := w_Index +1;
	
(*Temp L2 Warning*)		AddError[w_Index](
		b_ErrorTrig			:= get.events.b_TemperatureHighPhase[phases.L2],
		out_ST_Error			:= a_ActiveEvents[w_Index],
		w_ErrorID					:= 2,
		s_Message				:= 'high temperature L2 warning',
		e_sev					:= eseverity.Warning,
		b_AutoClear			:= TRUE,
	);
	w_Index := w_Index +1;
	
(*Temp L3 Warning*)		AddError[w_Index](
		b_ErrorTrig			:= get.events.b_TemperatureHighPhase[phases.L3],
		out_ST_Error			:= a_ActiveEvents[w_Index],
		w_ErrorID					:= 3,
		s_Message				:= 'high temperature L3 warning',
		e_sev					:= eseverity.Warning,
		b_AutoClear			:= TRUE,
	);
	w_Index := w_Index +1;
	
(*Temp L1 Alarm*)		AddError[w_Index](
		b_ErrorTrig			:= get.events.b_TemperatureTooHighPhase[phases.L1],
		out_ST_Error			:= a_ActiveEvents[w_Index],
		w_ErrorID					:= 4,
		s_Message				:= 'high temperature L1 alarm',
		e_sev					:= eseverity.Normalshutdown,
		t_TriggerTime		:= INT_TO_TIME(st_params.ui_TemperatureHighTripDelay*1000)
	);
	w_Index := w_Index +1;
	
(*Temp L2 Alarm*)		AddError[w_Index](
		b_ErrorTrig			:= get.events.b_TemperatureTooHighPhase[phases.L2],
		out_ST_Error			:= a_ActiveEvents[w_Index],
		w_ErrorID					:= 5,
		s_Message				:= 'high temperature L2 alarm',
		e_sev					:= eseverity.Normalshutdown,
		t_TriggerTime		:= INT_TO_TIME(st_params.ui_TemperatureHighTripDelay*1000)
	);
	w_Index := w_Index +1;
	
(*Temp L3 Alarm*)		AddError[w_Index](
		b_ErrorTrig			:= get.events.b_TemperatureTooHighPhase[phases.L3],
		out_ST_Error			:= a_ActiveEvents[w_Index],
		w_ErrorID					:= 6,
		s_Message				:= 'high temperature L3 alarm',
		e_sev					:= eseverity.Normalshutdown,
		t_TriggerTime		:= INT_TO_TIME(st_params.ui_TemperatureHighTripDelay*1000)
	);
	w_Index := w_Index +1;
	
(*Volt unbal Alarm*)	AddError[w_Index](
		b_ErrorTrig			:= get.events.b_VoltageUnbalanceTooHigh,
		out_ST_Error			:= a_ActiveEvents[w_Index],
		w_ErrorID					:= 7,
		s_Message				:= 'voltage unbalance fault',
		e_sev					:= eseverity.Normalshutdown,
		t_TriggerTime		:= INT_TO_TIME(st_params.ui_VoltageUnbalanceTripDelay*1000)
	);
	w_Index := w_Index +1;
	
(*Volt unbal Warning*)	AddError[w_Index](
		b_ErrorTrig			:= get.events.b_VoltageUnbalanceHigh,
		out_ST_Error			:= a_ActiveEvents[w_Index],
		w_ErrorID					:= 8,
		s_Message				:= 'voltage unbalance warning',
		e_sev					:= eseverity.Warning,
		b_AutoClear			:= TRUE
	);
	w_Index := w_Index +1;
	
(*OverCurr Alarm*)		AddError[w_Index](
		b_ErrorTrig			:= get.events.b_NeutralCurrentTooHigh,
		out_ST_Error			:= a_ActiveEvents[w_Index],
		w_ErrorID					:= 9,
		s_Message				:= 'Neutral current too high alarm',
		e_sev					:= eseverity.Normalshutdown,
		t_TriggerTime		:= T#10s
	);
	w_Index := w_Index +1;
	
(*Overcurr Warning*)	AddError[w_Index](
		b_ErrorTrig			:= get.events.b_NeutralCurrentHigh,
		out_ST_Error			:= a_ActiveEvents[w_Index],
		w_ErrorID					:= 10,
		s_Message				:= 'Neutral current high warning',
		e_sev					:= eseverity.Warning,
		b_AutoClear			:= TRUE
	);
	w_Index := w_Index +1;
END_METHOD

METHOD GetWearCounters : BOOL
VAR_INST
	//tof_ZPTOverload			:	tof := (pt := 5m);
	ZPTOverloadTripCount		:	FB_Varlogger;
	ZPTTempTripCount			:	FB_Varlogger;
END_VAR

ZPTOverloadTripCount(		TriggerInput := get.events.b_NeutralCurrentTooHigh, 
							LogItemGroup :=  eLogItemGroupID.ZPT, 
							LogItemName := 'ZptOvercurrentTripCnt', 
							LogType := eLogtypes.TrackCycles);

ZPTTempTripCount(			TriggerInput := get.events.b_TemperatureTooHighPhase[1] or  get.events.b_TemperatureTooHighPhase[2] or  get.events.b_TemperatureTooHighPhase[3], 
							LogItemGroup :=  eLogItemGroupID.ZPT, 
							LogItemName := 'ZptTempTripCnt', 
							LogType := eLogtypes.TrackCycles);
END_METHOD

METHOD Reset : BOOL

Reset := true;
END_METHOD

END_FUNCTION_BLOCK

// ---- POUs/Objects/NeutralTransformer/FB_NeutralTransformer_IO.TcPOU
FUNCTION_BLOCK INTERNAL FB_NeutralTransformer_IO
VAR	
	ZPT_read							AT %I* : ARRAY [1..3] OF ST_AnalogInputData;
END_VAR

VAR_OUTPUT
	r_TemperaturePhase							   : ARRAY [1..3] OF REAL;
	b_TemperatureOutOfRange							: BOOL;		
END_VAR

VAR_INPUT
	b_ResetOverCurrentProtection				:	BOOL;
END_VAR

r_TemperaturePhase[1] := EL320xToReal(i_In:=ZPT_Read[1].Value);
r_TemperaturePhase[2] := EL320xToReal(i_In:=ZPT_Read[2].Value);
r_TemperaturePhase[3] := EL320xToReal(i_In:=ZPT_Read[3].Value);
b_TemperatureOutOfRange:= ZPT_Read[1].Status.Overrange OR
	ZPT_Read[2].Status.Overrange OR
	ZPT_Read[3].Status.Overrange OR
	ZPT_Read[1].Status.Underrange OR
	ZPT_Read[2].Status.Underrange OR
	ZPT_Read[3].Status.Underrange;

METHOD PRIVATE EL320xToReal : REAL
VAR_INPUT
	i_In					: INT;
END_VAR
EL320xToReal:= TO_REAL(i_In) /10;
END_METHOD

END_FUNCTION_BLOCK

// ---- POUs/Functions-FBs-Programs/_generalFunctions/LimitTrigger.TcPOU
FUNCTION LimitTrigger : BOOL
VAR_INPUT
	r_HighLimit				: REAL := 0;
	r_HighWarning			: REAL := 0;
	b_HighEnable			: BOOL := FALSE;
	r_LowLimit				: REAL := 0;
	r_LowWarning			: REAL := 0;
	b_LowEnable				: BOOL := FALSE;
	r_Hysteresis			: REAL := 0;
END_VAR

VAR_IN_OUT CONSTANT
	r_In					: REAL;
END_VAR

VAR_OUTPUT
	b_Warning				: BOOL;
	b_Fault					: BOOL;
END_VAR

IF b_HighEnable THEN
	IF r_IN >= r_HighLimit THEN
		b_Fault := TRUE;
	ELSIF r_IN < (r_HighLimit - r_Hysteresis) THEN
		b_fault := FALSE;
	END_IF
	IF r_IN >= r_HighWarning THEN
		b_warning := TRUE;
	ELSIF r_IN < (r_HighWarning - r_Hysteresis) THEN
		b_warning := FALSE;
	END_IF

END_IF

IF b_LowEnable THEN
	IF r_IN <= r_LowLimit THEN
		b_fault := TRUE;
	ELSIF r_IN > (r_LowLimit + r_Hysteresis) THEN
		b_fault := FALSE;
	END_IF
	IF r_IN <= r_LowWarning THEN
		b_warning := TRUE;
	ELSIF r_IN > (r_LowWarning + r_Hysteresis) THEN
		b_warning:= FALSE;
	END_IF
END_IF

END_FUNCTION

// ---- POUs/Objects/CoolingSystem/FB_CoolingSystem.TcPOU
FUNCTION_BLOCK FB_CoolingSystem IMPLEMENTS ITF_standardFB
VAR_IN_OUT
	st_params					: ST_Coolingsystem_params;
END_VAR

VAR
	EMstopActive	:	Bool;	

	Heatpump 	: 	ITF_Heatpump;
	LGHeatpump	:	FB_LGThermaV;
	RemoteIO	:	FB_TruCompTCME21_IOModule;
	
	b_PumpEnable		AT %Q* : Bool;
	b_HeatpumpEnable	AT %Q* : Bool;
	b_HeatpumpFuseFB	AT %I* : Bool;
	
	
END_VAR


VAR_INPUT
	//Internal power supply status
	b_HVDC_Available			:	BOOL;	//from FB_ips, 24V online
	b_400v_Available 			:	BOOL;	//from FB_ips, 400vac online

	InverterConditioningRequirement		:	eConditioningRequirement;	
	BMSConditioningRequirement			:	eConditioningRequirement;
	EnclosureConditioningRequirement	:	eConditioningRequirement;
	ACDCConditioningRequirement			:	eConditioningRequirement;
	ManualConditioningRequirement		:	eConditioningRequirement;		
END_VAR

VAR_OUTPUT
	get						: st_CoolingSystem_Get;
	IPSRequest 				: ST_InternalPowerSupply_PowerDemand;//to FB_IPS, power requirements for cooling system
	b_FanPowerstackEnable	: BOOL;
END_VAR


Heatpump := LGHeatpump;
pumpcontrol();
HeatpumpControl();

RemoteIO();
RemoteIO.set.IPAddress 		:= st_params.IO_IPaddress;
get.r_CoolantTemperature 	:= RemoteIO.Get.AnalogInput1;
get.r_CoolantPressure		:=	Remoteio.Get.AnalogInput2;

IF not EMstopActive THEN
	IF Heatpump.HeatpumpState = eHeatpumpstate.Active_Cooling THEN
		get.CoolingSystemState := eCoolingSystemState.ActiveCooling;
	ELSIF  Heatpump.HeatpumpState = eHeatpumpstate.Active_Heating THEN
		get.CoolingSystemState := eCoolingSystemState.ActiveHeating;
	ELSIF b_PumpEnable THEN
		get.CoolingSystemState := eCoolingSystemState.Circulating;
	ELSE
		get.CoolingSystemState := eCoolingSystemState.OFF;
	END_IF
end_if

{warning 'Add method implementation '}
METHOD EMstop : BOOL
EMstopActive := true;
Heatpump.EMstop();
get.CoolingSystemState := eCoolingSystemstate.EMSTOP;
EMstop := true;
END_METHOD

{warning 'Add method implementation '}
METHOD getDiagnostics
VAR_IN_OUT
	AddError		: ARRAY [*] OF FB_AddErrorST;
	a_ActiveEvents	: ARRAY [*] OF ST_ErrorStruct;
	w_Index			: WORD;
END_VAR
AddError[w_Index](
	b_ErrorTrig			:= get.events.b_CoolingSystemFuseFailure,
	out_ST_Error		:= a_ActiveEvents[w_Index],
	w_ErrorID			:= 1,
	e_ObjectID			:=  eObject_ID.Cooling,
	s_Message			:= 'Heatpump breaker tripped, heatpump inoperative',
	e_sev				:= eseverity.Warning,
	b_AutoClear			:= TRUE
);
w_Index := w_Index +1;
	

AddError[w_Index](
	b_ErrorTrig			:= Get.Events.b_CoolingLoopPressureTooLow,
	out_ST_Error		:= a_ActiveEvents[w_Index],
	w_ErrorID			:= 2,
	s_Message			:= 'pressure fault',
	e_sev				:= eSeverity.NormalShutdown,	
	b_AutoClear			:= FALSE,
);
w_Index := w_Index +1;	
	

AddError[w_Index](
	b_ErrorTrig			:= Get.Events.b_CoolingLoopPressureLow,
	out_ST_Error		:= a_ActiveEvents[w_Index],
	w_ErrorID			:= 3,
	s_Message			:= 'pressure warning',
	e_sev				:= eSeverity.Warning,	
	b_AutoClear			:= TRUE,
);
w_Index := w_Index +1;	
	
	
AddError[w_Index](
	b_ErrorTrig			:= get.events.b_CoolantTempHigh,
	out_ST_Error		:= a_ActiveEvents[w_Index],
	w_ErrorID			:= 4,
	s_Message			:= 'Coolant temperature high',
	e_sev				:= eseverity.warning,
	b_AutoClear			:= TRUE
);
w_Index := w_Index +1;
	

AddError[w_Index](
	b_ErrorTrig			:= get.events.b_CoolantTempTooHigh,
	out_ST_Error		:= a_ActiveEvents[w_Index],
	w_ErrorID			:= 5,
	s_Message			:= 'Coolant temperature too high',
	e_sev				:= eseverity.NormalShutdown,
);
w_Index := w_Index +1;


AddError[w_Index](
	b_ErrorTrig			:= get.events.b_CoolantTempLow,
	out_ST_Error		:= a_ActiveEvents[w_Index],
	w_ErrorID			:= 6,
	s_Message			:= 'Coolant temperature low',
	e_sev				:= eseverity.warning,
	b_AutoClear			:= TRUE
);
w_Index := w_Index +1;

Heatpump.getDiagnostics(AddError := AddError, a_ActiveEvents := a_ActiveEvents, w_Index := w_Index);
END_METHOD

METHOD HeatpumpControl : BOOL
VAR_INPUT
END_VAR


VAR_inst
	ton_heatpumpPowerDelay	:	Ton	:=	(PT := T#1s);
END_VAR
//if any of the mayor parts require conditioning, the heatpump is required and thus 400VAC is required
if not EMStopActive and 
	(InverterConditioningRequirement > eConditioningRequirement.Pumprequired OR 
	BMSConditioningRequirement > eConditioningRequirement.Pumprequired OR 
	ACDCConditioningRequirement > eConditioningRequirement.Pumprequired) or
	ManualConditioningRequirement > eConditioningRequirement.none then
	
	ipsrequest.b_Demand_400V := true;
	
	if b_400v_Available then
		if Heatpump.HeatpumpState >= eHeatpumpState.Standby then 
			if InverterConditioningRequirement = eConditioningRequirement.CoolingRequired or
				BMSConditioningRequirement = eConditioningRequirement.CoolingRequired OR 
				ACDCConditioningRequirement = eConditioningRequirement.CoolingRequired OR
				ManualConditioningRequirement = eConditioningRequirement.CoolingRequired then
					Heatpump.OperationMode := eHeatpumpMode.Cooling;
					Heatpump.Setpoint := max(main_fast.enclosure.get.climate.r_Dewpoint + 2, 18);
			elsif InverterConditioningRequirement = eConditioningRequirement.HeatingRequired or
				BMSConditioningRequirement = eConditioningRequirement.HeatingRequired OR 
				ACDCConditioningRequirement = eConditioningRequirement.HeatingRequired or
				ManualConditioningRequirement = eConditioningRequirement.HeatingRequired then
					Heatpump.OperationMode := eHeatpumpMode.Heating;
					Heatpump.Setpoint := 35;
			END_IF
		end_if
	end_if
else
	Heatpump.OperationMode := eHeatpumpMode.Standby;
	if heatpump.HeatpumpState <> eHeatpumpState.Active_Heating and heatpump.HeatpumpState <> eHeatpumpState.Active_cooling then
		ipsrequest.b_Demand_400V := false;
	END_IF
END_IF

ton_heatpumpPowerDelay(in := b_400v_Available and b_HeatpumpFuseFB);
b_HeatpumpEnable := ton_heatpumpPowerDelay.Q;
END_METHOD

{warning 'Add method implementation '}
METHOD Init : BOOL
Heatpump.Init();
END_METHOD

METHOD InternalConditioning : eConditioningRequirement
VAR_INST
	ManualconditioningTimelimit	:	ton := (PT := T#30M);
END_VAR

InternalConditioning := eConditioningrequirement.none;

// IF 		st_Params.b_ActivateCooling AND NOT ManualconditioningTimelimit.q 	or 
// 		
// 	THEN
// 	InternalConditioning := eConditioningrequirement.CoolingRequired;
// ELSIF st_Params.b_ActivateHeating AND NOT ManualconditioningTimelimit.q THEN
// 	InternalConditioning := eConditioningrequirement.HeatingRequired;
// END_IF
// 
// //to prevent the system being stuck in a manual mode. It is automatically deactivated after the set time limit (1H). 
// ManualConditioningTimelimit(in := st_Params.b_ActivateCooling OR st_Params.b_ActivateHeating);
END_METHOD

METHOD PumpControl : BOOL
VAR_INPUT
END_VAR

var_inst
	tof_PumpOffDelay	:	Tof	:=	(pt := T#30s);
	PumpRequired		:	Bool;
END_VAR

PumpRequired := InverterConditioningRequirement > eConditioningrequirement.none or
 				ACDCConditioningRequirement	 > eConditioningrequirement.none AND
				not EMstopActive and 
					ManualConditioningRequirement > eConditioningRequirement.none or
					(BMSConditioningRequirement > eConditioningrequirement.none or
					EnclosureConditioningRequirement > eConditioningrequirement.none);

tof_PumpOffDelay(in := PumpRequired);

IPSRequest.b_Demand_HVDC := PumpRequired or b_PumpEnable; 
b_PumpEnable := tof_PumpOffDelay.Q and b_HVDC_Available;


//enclosureconditioning requires powerstack fan to run
b_FanPowerstackEnable := EnclosureConditioningRequirement > eConditioningrequirement.none and b_PumpEnable;
END_METHOD

{warning 'Add method implementation '}
METHOD Reset : BOOL
EMstopActive := false;
Heatpump.Reset();

IF get.CoolingSystemState = eCoolingSystemstate.EMSTOP THEN
	get.CoolingSystemState := eCoolingSystemstate.OFF;
end_if

Reset := true;
END_METHOD

END_FUNCTION_BLOCK

// ---- POUs/Objects/CoolingSystem/FB_LGThermaV.TcPOU
FUNCTION_BLOCK FB_LGThermaV implements ItF_Heatpump

VAR
	ReadCoils		:	FB_MBReadCoils;
	ReadInputs		:	FB_MBReadInputs;
	Readregs		:	FB_MBReadregs;
	ReadInputRegs	:	FB_MBReadInputRegs;
	WriteCoils		:	FB_MBWriteCoils;
	WriteRegs		:	FB_MBWriteRegs;
	
END_VAR

VAR_OUTPUT
	Get				:	st_heatpump_Get;
END_VAR

VAR_IN_OUT CONSTANT
	st_params		: 	ST_Coolingsystem_params;
END_VAR

VAR_INPUT
	ACPowerStatus	:	BOOL;
	HeatPumpID		:	BYTE;
END_VAR
		
VAR
	ton_MBBUSYTimeOut		: TON := (PT := T#10s);
	DataBuffer				:	ARRAY[0..50] OF WORD;
	Ton_ErrorTimer			:	Ton := (PT := T#5M);
	MBRetryCount			:	BYTE;
	TransmissionDone		:	F_Trig;
	CommIntervalTimer		:	Ton	:=	(PT := T#5S);
END_VAR

VAR
	b_EMStop						:	BOOL;
	b_resetErrors					:	BOOL;
	sPressureErrorText				:	STRING;
	sCompressorErrorText			:	STRING;
	sPumpErrorText					:	STRING;
	sWaterTempErrorText				:	STRING;
	
	Coils		: 	LG_Coils;
	Inputs 		: 	LG_Inputregs;
	Statusbits	:	LG_StatusBits;
	ControlRegs	:	LG_Controlregs;
END_VAR

VAR
	CoilStatus		:	BYTE;

	RequestedOperationMode	:	eHeatpumpMode;
	RequestedSetpoint		:	Real;

	HeatpumpEMOperationAvailable	:	Bool;
END_VAR

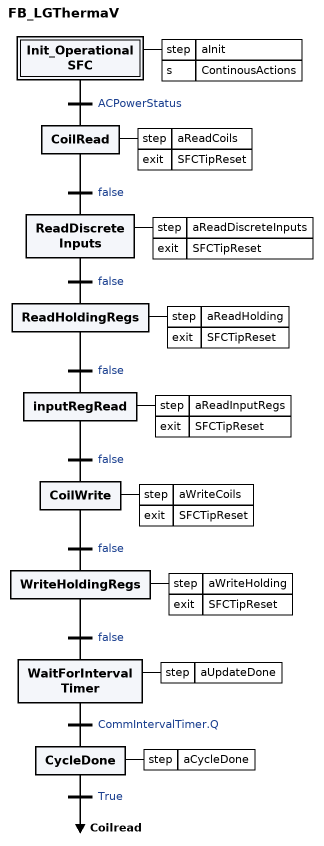
INITIAL_STEP Init_OperationalSFC:
    aInit(N);  // step action
    ContinousActions(s);
END_STEP
TRANSITION FROM Init_OperationalSFC TO CoilRead
    := ACPowerStatus;
END_TRANSITION
STEP CoilRead:
    aReadCoils(N);  // step action
    SFCTipReset(P0);  // exit action
END_STEP
TRANSITION FROM CoilRead TO ReadDiscreteInputs
    := false;
END_TRANSITION
STEP ReadDiscreteInputs:
    aReadDiscreteInputs(N);  // step action
    SFCTipReset(P0);  // exit action
END_STEP
TRANSITION FROM ReadDiscreteInputs TO ReadHoldingRegs
    := false;
END_TRANSITION
STEP ReadHoldingRegs:
    aReadHolding(N);  // step action
    SFCTipReset(P0);  // exit action
END_STEP
TRANSITION FROM ReadHoldingRegs TO inputRegRead
    := false;
END_TRANSITION
STEP inputRegRead:
    aReadInputRegs(N);  // step action
    SFCTipReset(P0);  // exit action
END_STEP
TRANSITION FROM inputRegRead TO CoilWrite
    := false;
END_TRANSITION
STEP CoilWrite:
    aWriteCoils(N);  // step action
    SFCTipReset(P0);  // exit action
END_STEP
TRANSITION FROM CoilWrite TO WriteHoldingRegs
    := false;
END_TRANSITION
STEP WriteHoldingRegs:
    aWriteHolding(N);  // step action
    SFCTipReset(P0);  // exit action
END_STEP
TRANSITION FROM WriteHoldingRegs TO WaitForIntervalTimer
    := false;
END_TRANSITION
STEP WaitForIntervalTimer:
    aUpdateDone(N);  // step action
END_STEP
TRANSITION FROM WaitForIntervalTimer TO CycleDone
    := CommIntervalTimer.Q;
END_TRANSITION
STEP CycleDone:
    aCycleDone(N);  // step action
END_STEP
TRANSITION FROM CycleDone TO Coilread
    := True;
END_TRANSITION

ACTION aCycleDone:
CommIntervalTimer.IN := false;
END_ACTION

ACTION aInit:
get.HeatPumpState := eHeatpumpstate.OFF;
SFCReset := FALSE;
get.Events.b_CommWarning := FALSE;
MBRetryCount := 0;
END_ACTION

ACTION aReadCoils:
CommIntervalTimer.IN := TRUE;

TransmissionDone(clk := ReadCoils.bBusy);

ReadCoils(sIPAddr	:=	st_params.IO_IPaddress,
						nTCPPort	:=	502,
						nUnitID 	:=  HeatpumpID,
						nQuantity 	:= 	5,
						nMBAddr		:=	0,
						cbLength 	:= 	6,
						pDestAddr	:=	ADR(CoilStatus),
						tTimeout	:=	T#100ms,//st_params.t_ModbusTimeOut,
						bExecute	:=	NOT (ReadCoils.bbusy OR TransmissionDone.Q),
				);
	

IF TransmissionDone.q THEN
	IF NOT ReadCoils.bError THEN
		//Full datastruct for debug purposes. Can be removed later
		Coils.b_EnableOperation := CoilStatus.0;
		Coils.b_EnableSwwOperation := CoilStatus.1;
		Coils.b_EnableSilentMode := CoilStatus.2;
		Coils.b_EnableDesinfectionMode := Coilstatus.3;
		Coils.b_EmstopActive := CoilStatus.4;
		Coils.b_EnableEmStop := CoilStatus.5;
		//Full datastruct for debug purposes. Can be removed later
		
	ELSE
		MBRetryCount := MBRetryCount + 1;
	END_IF
	
	sfctip := TRUE;
END_IF
END_ACTION

ACTION aReadDiscreteInputs:
TransmissionDone(clk := Readinputs.bBusy);

Readinputs(				sIPAddr		:=	st_params.IO_IPaddress,
						nTCPPort	:=	502,
						nUnitID 	:= 	HeatpumpID,
						nQuantity 	:= 	16,
						nMBAddr		:=	0,
						cbLength 	:= 	SIZEOF(Databuffer),
						pDestAddr	:=	ADR(Databuffer),
						tTimeout	:=	T#100ms,//st_params.t_ModbusTimeOut,
						bExecute	:=	NOT (Readinputs.bbusy OR TransmissionDone.Q),
				);


IF TransmissionDone.q THEN
	IF NOT ReadInputs.bError THEN
		//Full datastruct for debug purposes. Can be removed later
		Statusbits.b_WaterFlowNOK := DataBuffer[0].0;
		Statusbits.b_WaterPumpOn := DataBuffer[0].1;
		Statusbits.b_ExtWaterPumpOn := DataBuffer[0].2;
		Statusbits.b_CompressorOn := DataBuffer[0].3;
		Statusbits.b_DefrostOn := DataBuffer[0].4;
		Statusbits.b_SWWModeOn := DataBuffer[0].5;
		Statusbits.b_SWWTankDesinfectionActive := DataBuffer[0].6;
		Statusbits.b_SilentModeOn := DataBuffer[0].7;
		Statusbits.b_CoolingActive := DataBuffer[0].8;
		Statusbits.b_SolarPumpActive := DataBuffer[0].9;
		Statusbits.b_BackupHeater1Active := DataBuffer[0].10;
		Statusbits.b_BackupHeater2Active := DataBuffer[0].11;
		Statusbits.b_SWWBoostHeaterActive := DataBuffer[0].12;
		Statusbits.b_ErrorActive := DataBuffer[0].13;
		Statusbits.b_EMOperationAvailable := DataBuffer[0].14;
		Statusbits.b_EMSWWOperationAvailable := DataBuffer[0].15;
		Statusbits.b_MixPumpActive := DataBuffer[1].0;
		//Full datastruct for debug purposes. Can be removed later
		
		get.Events.b_PumpError := DataBuffer[0].0;
		get.events.b_DefrostingActive := DataBuffer[0].4;
		
		
		//error active and no em operation allowed
		IF DataBuffer[0].13 THEN
			get.HeatPumpState := eHeatpumpstate.ERROR;
			IF NOT DataBuffer[0].14 THEN
				HeatpumpEMOperationAvailable := FALSE;
			ELSE
				HeatpumpEMOperationAvailable := TRUE;
			END_IF
		ELSIF get.HeatPumpState = eHeatpumpstate.ERROR THEN
			get.HeatPumpState := eHeatpumpstate.Initializing;
			HeatpumpEMOperationAvailable := FALSE;
		END_IF
		
		//done, preset for next step
		MBRetryCount := 0;
	ELSE
		MBRetryCount := MBRetryCount + 1;
	END_IF
	sfctip := TRUE;
END_IF
END_ACTION

ACTION aReadHolding:
TransmissionDone(clk := Readregs.bBusy);

Readregs(	sIPAddr		:=	st_params.IO_IPaddress,
			nTCPPort	:=	502,
			nUnitID 	:= 	HeatpumpID,
			nQuantity 	:= 	10,
			nMBAddr		:=	0,
			cbLength 	:= 	SIZEOF(Databuffer),
			pDestAddr	:=	ADR(Databuffer),
			tTimeout	:=	T#100ms,//st_params.t_ModbusTimeOut,
			bExecute	:=	NOT (ReadRegs.bbusy OR TransmissionDone.Q),
		);


IF TransmissionDone.q THEN
	IF NOT Readregs.bError THEN
		Controlregs.ui_OperatingMode := Databuffer[0];
		Controlregs.ui_ControlMode := Databuffer[1];
		Controlregs.r_Setpoint1 := (WORD_TO_REAL(Databuffer[2])/10);
		Controlregs.r_RoomSetpoint := (WORD_TO_REAL(Databuffer[3])/10);
		Controlregs.ui_TempShiftValue := Databuffer[4];
		Controlregs.r_Setpoint2 := (WORD_TO_REAL(Databuffer[5])/10);
		Controlregs.r_RoomSetpoint2 := (WORD_TO_REAL(Databuffer[6])/10);
		Controlregs.ui_TempShiftValue2 := Databuffer[7];
		Controlregs.r_DHWgoalTemp := (WORD_TO_REAL(Databuffer[8])/10);
		Controlregs.ui_EnergyStatus := Databuffer[9];
		
		get.Setpoint := (WORD_TO_REAL(Databuffer[2])/10);


		IF get.HeatPumpState <> eHeatpumpstate.ERROR THEN
			CASE get.HeatPumpState OF
				0:
					get.HeatPumpState := eHeatpumpstate.Standby;
				1:
					get.HeatPumpState := eHeatpumpstate.Active_Cooling;
				2:
					get.HeatPumpState := eHeatpumpstate.Active_Heating;
			END_CASE
		END_IF
	
		//done, preset for next step
		MBRetryCount := 0;

	ELSE
		MBRetryCount := MBRetryCount + 1;
		
	END_IF
	sfctip := TRUE;
END_IF
END_ACTION

ACTION aReadInputRegs:
TransmissionDone(clk := ReadInputregs.bBusy);

ReadInputregs(	sIPAddr		:=	st_params.IO_IPaddress,
				nTCPPort	:=	502,
				nUnitID 	:= 	HeatpumpID,
				nQuantity 	:= 	14,
				nMBAddr		:=	0,
				cbLength 	:= 	SIZEOF(Databuffer),
				pDestAddr	:=	ADR(Databuffer),
				tTimeout	:=	T#100ms,//st_params.t_ModbusTimeOut,
				bExecute	:=	NOT (ReadInputRegs.bbusy OR TransmissionDone.Q),
		);


IF TransmissionDone.q THEN
	IF NOT ReadInputregs.bError THEN		
	//Full datastruct for debug purposes. Can be removed later
		Inputs.UI_ErrorCode := Databuffer[0];	
		Inputs.ui_OperationalMode := (Databuffer[1]);	
		Inputs.r_CoolantInletTemp := WORD_TO_REAL((Databuffer[2]))/10;	
		Inputs.r_CoolantOutletTemp := WORD_TO_REAL((Databuffer[3]))/10;
		Inputs.r_BackupHeaterTemp := WORD_TO_REAL((Databuffer[4]))/10;
		Inputs.r_SWWTankTemp :=  WORD_TO_REAL((Databuffer[5]))/10;
		Inputs.r_SolarCollectorTemp := WORD_TO_REAL((Databuffer[6]))/10;
		Inputs.r_RoomTemp1 := WORD_TO_REAL((Databuffer[7]))/10;
		Inputs.r_FlowRate := WORD_TO_REAL((Databuffer[8]))/10;
		Inputs.r_FlowTempCircuit2 := WORD_TO_REAL((Databuffer[9]))/10;
		Inputs.r_RoomTemp2 := WORD_TO_REAL((Databuffer[10]))/10;
		Inputs.UI_EnergyStatus := (Databuffer[11]);
		Inputs.r_OutsideTemp := WORD_TO_REAL((Databuffer[12]))/10;
		Inputs.r_CoolantPressure := WORD_TO_REAL((Databuffer[13]))/10;
	//full datastruct for debug purposes. can be removed later	
	ELSE
		MBRetryCount := MBRetryCount + 1;
	END_IF
	sfctip := TRUE;
END_IF
END_ACTION

ACTION aUpdateDone:
SFCTip := FALSE;
END_ACTION

ACTION aWriteCoils:


CoilStatus.0 := requestedOperationMode <> eHeatpumpMode.Standby; // operation off

CoilStatus.5 := EMHeatingModeRequired();



TransmissionDone(clk := WriteCoils.bBusy);

WriteCoils		(sIPAddr	:=	st_params.IO_IPaddress,
				nTCPPort	:=	502,
				nUnitID 	:= 	HeatpumpID,
				nQuantity 	:= 	5,
				nMBAddr		:=	0,
				cbLength 	:= 	1,
				pSrcAddr	:=	ADR(CoilStatus),
				tTimeout	:=	T#100ms,
				bExecute	:=	NOT (WriteCoils.bbusy OR TransmissionDone.Q),
		);
	

IF TransmissionDone.q THEN
	IF NOT WriteCoils.bError THEN
			sfctip := TRUE;
			
		ELSE
			MBRetryCount := MBRetryCount + 1;
			sfctip := NOT sfctip;
		END_IF
	END_IF
//ELSE
//	sfctip := NOT sfctip;
//END_IF
END_ACTION

ACTION aWriteHolding:

